FUNCTION_BLOCK "KebaHT4"	// FB 80
TITLE = Maintenance Control HT4
//
//COPYRIGHT:    (C) 1999 BY  BUEHLER AG
//                           CH-9240 UZWIL  SWITZERLAND
//
//PRODUCT:      
//
//TITLE:        MAINTENANCE MOTOR CONTROL "HT4"
//
//              LOKALE MOTOREN STEUERUNG "HT4"
//
//---------------------------------------------------------------------------
//
//IDENT:        AUTHOR:             DEPT:                         DATE:
//
//FB80.1A       S. Kalberer         CT3                           14.04.1999
//              Generated by S5/S7 Converter
//              Adjusted from S5 FB180.2C and DB180.2A
//              Outputs > 511 will set the Peripherial Output (PA) directly
//---------------------------------------------------------------------------
//
//PURPOSE:      - DATA TRANSFER BETWEEN HT4 AND PLC, VIA DB80
//
//                REMARK: ALL PASSWORD PROTECTED FUNCTIONS ARE MARKED WITH *
//
//RESTRICTIONS: - S7
//
//                !!! IMPORTANT !!!
//              - FB80 MUST BE CALLED AFTER FC9 IN OB1, TO PROCESS THE
//                OUTPUTS PROPELRY!!!
//
//              - FOLLOWING DB's MUST BE AVAILABLE:
//                . DB80 = Instance DB - COMMUNICATION BUFFER HT4 - PLC 
//                . DB81 = REFERENCE TABLE MOTORS (M)
//                . DB82 = REFERENCE TABLE VARIOUS ELEMENTS (V, FC, etc.)
//
//                . A DIGITAL OUTPUT FROM 128.0 TO 255.7 WILL BE PROCESSED
//                  INDIRECT VIA THE DB DEFINED IN DB80, DW63. THE RELEVANT
//                  DB AND DW IN THIS DB MUST BE AVAILABLE.
//                  (DW-No.IN DB = OUTPUT-BYTE-No.)
//
//              - IF THE NUMBER OF DW/OBJECT IS CHANGED, THE PARAMETERS (!@) 
//                HAVE TO BE CHANGED ACCORDINGLY !
//
//---------------------------------------------------------------------------
//$EJECT
//STRUCTURE:
//==========
//OB1:
//   | --> FC9: Call Groups
//   |
//   | --> FC80: Call Groups
//   |          |
//              |
//              | --> FB80: (REMOTE CONTROL), DB80: (COMM-BUFFER HT4 - PLC)
//                         |
//                         | --> e.g. DB81: (REF-TABLE MOTORS)
//                         |     (see Par_Motor_DBNo)
//                         | --> e.g. DB82: (REF-TABLE VARIOUS ELEMENTS)
//                         |     (see Par_Variousr_DBNo)
//       
//
//PARAMETERS and VARIABLES:
//=========================
//
//DBW 104 VAR.Errror
//  +0.0 = Error.
//  +1.0 = Error.
//  +1.1 = Error.Cfg_Fault    
//  +1.2 = Error.Obj_NoNull  
//  +1.3 = Error.Obj_Not_Found  
//  +1.4 = Error.Invalid_Password        
//  +1.5 = Error.Machine_Stop            
//  +1.6 = Error.Comm_Timeout   
//  +1.7 = Error.Summary                 
//
//DBW 106 VAR.Info
//  +0.0 = Info.Obj_Ready
//  +0.1 = Info.
//  +0.2 = Info.
//  +0.3 = Info.Obj_DO1_Set
//  +0.4 = Info.Obj_DO2_Set
//  +0.5 = Info.Obj_DO3_Set
//  +0.6 = Info.Obj_DO4_Set
//  +0.7 = Info.Obj_AO1_Set
//
//  +1.0 = Info.HT4_Enabled 
//  +1.1 = Info.HT4_Service_Mode
//  +1.2 = Info.HT4_password_ok 
//  +1.3 = Info.                
//  +1.4 = Info.                
//  +1.5 = Info.                
//  +1.6 = Info.HT4_KeyPressedFlag
//  +1.7 = Info.HT4_KeyPressedEdge
//
//DBW 108 Err_Invalid_ObjNo
//
//DBW 110 VAR_Actual_OjbNo                \
//DBW 112 VAR_DO1_ByteAddr                 | 
//DBW 114 VAR_DO1_BitAddr                  | copy from reference DB
//DBW 116 VAR_DO2_ByteAddr                 |
//DBW 118 VAR_DO2_BitAddr                  | 
//DBW 120 VAR_DO3_ByteAddr                 |
//DBW 122 VAR_DO3_BitAddr                  | 
//DBW 124 VAR_DO4_ByteAddr                 |
//DBW 126 VAR_DO4_BitAddr                  | 
//DBW 128 VAR_AO1_ByteAddr                 | 
//DBW 130 VAR_ObjState                     | 
//  +0.0 = spare                           /
//  +1.0 = ManMode
//  +1.1 = DO1_Set
//  +1.2 = DO2_Set
//  +1.3 = DO3_Set
//  +1.4 = DO4_Set
//  +1.5 = AO1_Set
//  +1.6 = 
//  +1.7 = 
//
//DBW 132 = 0    Par_AO1 Man Mode Value
//
//DBW 134 = 81  Par_Motor DB Number
//
//DBW 136 = 82  Par_Various DB Number
//
//(!@)
//DBW 138 = 0    Par_ObjDB_1stBlockOff: Byte Offset (Start oft first block)
//
//(!@)
//DBW 140 = 22   Par_ObjDB_BlockLength: Block length (Byte)
//
AUTHOR : SK
FAMILY : KebaHT4
NAME : HT4
VERSION : 1.0
VAR
  KeyStatus : STRUCT 	//Key Status
   InternalCode : BYTE ;
   UserCode : BYTE ;
   Char_8 : BOOL ;
   Char_9 : BOOL ;
   Char_A : BOOL ;
   Char_Esc : BOOL ;	//'B: esc'
   Char_C : BOOL ;
   Char_D : BOOL ;
   Char_E : BOOL ;
   Char_F : BOOL ;
   Char_F1 : BOOL ;	//'0: F1'
   Char_F2 : BOOL ;	//'1: F2'
   Char_F3 : BOOL ;	//'2: F3'
   Char_F4 : BOOL ;	//'3: F4'
   Char_F5 : BOOL ;	//'4: F5'
   Char_F6 : BOOL ;	//'5: F6'
   Char_F7 : BOOL ;	//'6: F7'
   Char_F8 : BOOL ;	//'7: F8'
   Char_O : BOOL ;
   Char_P : BOOL ;
   Char_Q : BOOL ;
   Char_R : BOOL ;
   Char_Alt : BOOL ;	//'S: Alt'
   Char_T : BOOL ;
   Char_U : BOOL ;
   Char_Start : BOOL ;	//'V: Start'
   Char_G : BOOL ;
   Char_H : BOOL ;
   Char_I : BOOL ;
   Char_J : BOOL ;
   Char_K : BOOL ;
   Char_L : BOOL ;
   Char_M : BOOL ;
   Char_N : BOOL ;
   EmergencyStop : BOOL ;
   EditModeActive : BOOL ;
   spare0602 : BOOL ;
   spare0603 : BOOL ;
   spare0604 : BOOL ;
   spare0605 : BOOL ;
   spare0606 : BOOL ;
   ActiveBit : BOOL ;
   Char_Ctrl : BOOL ;	//'W: Ctrl'
   Char_X : BOOL ;
   Char_Y : BOOL ;
   Char_Stop : BOOL ;	//'Z: Stop'
   Char_Shift : BOOL ;	//'[: Shift'
   Char_BackSlash : BOOL ;	//'\: '
   Char_SqBracketClos : BOOL ;	//']: '
   Char_Enter : BOOL ;	//'^: Enter'
  END_STRUCT ;
  EditLineNo : WORD ;	//EditLine No (HT4: 0..4)
  D_5 : WORD ;	// reserviert              ==>  S5
  D_6 : WORD ;	// reserviert              ==>  S5
  D_7 : WORD ;	// reserviert              ==>  S5
  D_8 : WORD ;	// reserviert              ==>  S5
  D_9 : WORD ;	// reserviert              <==  S5
  D_10 : WORD ;	// reserviert              <==  S5
  D_11 : WORD ;	// reserviert              <==  S5
  D_12 : WORD ;	// reserviert              <==  S5
  D_13 : WORD ;	// reserviert              <==  S5
  D_14 : WORD ;	// reserviert              <==  S5
  D_15 : WORD ;	//                         <==  S5
  DB_ID : ARRAY  [1 .. 8 ] OF CHAR ;
  LEDBitmap : STRUCT 	//LED Bitmap Red (only HT4)
   Char_8 : BOOL ;
   Char_9 : BOOL ;
   Char_A : BOOL ;
   Char_Esc : BOOL ;	//'B: esc'
   Char_C : BOOL ;
   Char_D : BOOL ;
   Char_E : BOOL ;
   Char_F : BOOL ;
   Char_F1 : BOOL ;	//'0: F1'
   Char_F2 : BOOL ;	//'1: F2'
   Char_F3 : BOOL ;	//'2: F3'
   Char_F4 : BOOL ;	//'3: F4'
   Char_F5 : BOOL ;	//'4: F5'
   Char_F6 : BOOL ;	//'5: F6'
   Char_F7 : BOOL ;	//'6: F7'
   Char_F8 : BOOL ;	//'7: F8'
   Char_O : BOOL ;
   Char_P : BOOL ;
   Char_Q : BOOL ;
   Char_R : BOOL ;
   Char_Alt : BOOL ;	//'S: Alt'
   Char_T : BOOL ;
   Char_U : BOOL ;
   Char_Start : BOOL ;	//'V: Start'
   Char_G : BOOL ;
   Char_H : BOOL ;
   Char_I : BOOL ;
   Char_J : BOOL ;
   Char_K : BOOL ;
   Char_L : BOOL ;
   Char_M : BOOL ;
   Char_N : BOOL ;
   TestOutput : BOOL ;
   SpaceLine : BOOL ;
   spare0402 : BOOL ;
   spare0403 : BOOL ;
   spare0404 : BOOL ;
   ReleaseKeyclick : BOOL ;
   DepressKeyclick : BOOL ;
   Beep : BOOL ;
   Char_Ctrl : BOOL ;	//'W: Ctrl'
   Char_X : BOOL ;
   Char_Y : BOOL ;
   Char_Stop : BOOL ;	//'Z: Stop'
   Char_Shift : BOOL ;	//'[: Shift'
   Char_BackSlash : BOOL ;	//'\: '
   Char_SqBracketClos : BOOL ;	//']: '
   Char_Enter : BOOL ;	//'^: Enter'
  END_STRUCT ;
  LEDFlashmap : STRUCT 	//LED Flashmap Red (only HT4)
   Char_8 : BOOL ;
   Char_9 : BOOL ;
   Char_A : BOOL ;
   Char_Esc : BOOL ;	//'B: esc'
   Char_C : BOOL ;
   Char_D : BOOL ;
   Char_E : BOOL ;
   Char_F : BOOL ;
   Char_F1 : BOOL ;	//'0: F1'
   Char_F2 : BOOL ;	//'1: F2'
   Char_F3 : BOOL ;	//'2: F3'
   Char_F4 : BOOL ;	//'3: F4'
   Char_F5 : BOOL ;	//'4: F5'
   Char_F6 : BOOL ;	//'5: F6'
   Char_F7 : BOOL ;	//'6: F7'
   Char_F8 : BOOL ;	//'7: F8'
   Char_O : BOOL ;
   Char_P : BOOL ;
   Char_Q : BOOL ;
   Char_R : BOOL ;
   Char_Alt : BOOL ;	//'S: Alt'
   Char_T : BOOL ;
   Char_U : BOOL ;
   Char_Start : BOOL ;	//'V: Start'
   Char_G : BOOL ;
   Char_H : BOOL ;
   Char_I : BOOL ;
   Char_J : BOOL ;
   Char_K : BOOL ;
   Char_L : BOOL ;
   Char_M : BOOL ;
   Char_N : BOOL ;
   spare0400 : BOOL ;
   spare0401 : BOOL ;
   spare0402 : BOOL ;
   spare0403 : BOOL ;
   spare0404 : BOOL ;
   spare0405 : BOOL ;
   spare0406 : BOOL ;
   spare0407 : BOOL ;
   Char_Ctrl : BOOL ;	//'W: Ctrl'
   Char_X : BOOL ;
   Char_Y : BOOL ;
   Char_Stop : BOOL ;	//'Z: Stop'
   Char_Shift : BOOL ;	//'[: Shift'
   Char_BackSlash : BOOL ;	//'\: '
   Char_SqBracketClos : BOOL ;	//']: '
   Char_Enter : BOOL ;	//'^: Enter'
  END_STRUCT ;
  TextNo_Line0 : INT ;	// Textnummer Zeile 0      <==  S5
  TextNo_Line1 : INT ;	// Textnummer Zeile 1      <==  S5
  TextNo_Line2 : INT ;	// Textnummer Zeile 2      <==  S5
  TextNo_Line3 : INT ;	// Textnummer Zeile 3      <==  S5
  D_30 : WORD ;	// reserviert              <==  S5
  D_31 : WORD ;	// reserviert              <==  S5
  D_32 : WORD ;	// reserviert              <==  S5
  D_33 : WORD ;	// reserviert              <==  S5
  D_34 : WORD ;	// Variable                <==  S5
  D_35 : WORD ;	// Variable                <==  S5
  D_36 : WORD ;	// Variable                <==  S5
  D_37 : WORD ;	// Variable                <==  S5
  D_38 : WORD ;	// Variable                <==  S5
  HT4_Inp_Password : WORD ;	// HT4.var_inp_password    <==  S5
  HT4_Target_ObjNo : WORD ;	// HT4.var_target_object_no<==> S5
  HT4_Actual_ObjNo : WORD ;	// HT4.var_actual_object_no<==> S5
  D_42 : WORD ;	// Variable                <==> S5
  D_43 : WORD ;	// Variable                <==> S5
  D_44 : WORD ;	// Variable                <==> S5
  D_45 : WORD ;	// Variable                <==> S5
  D_46 : WORD ;	// Variable                <==> S5
  D_47 : WORD ;	// Variable                <==> S5
  D_48 : WORD ;	// Variable                <==> S5
  D_49 : WORD ;	// Variable                <==> S5
  D_50 : WORD ;	// ________________________________
  D_51 : WORD ;	// ==<INTERNAL USED VARIABLES>=====
  Error : STRUCT 	// VAR.error_word
   spare0000 : BYTE ;
   spare0100 : BOOL ;
   Cfg_Fault : BOOL ;
   Obj_NoNull : BOOL ;
   Obj_NotFound : BOOL ;
   Invalid_Password : BOOL ;
   Machine_Stop : BOOL ;
   Comm_Timeout : BOOL ;
   Summary : BOOL ;
  END_STRUCT ;
  Info : STRUCT 	// VAR.info_word
   Obj_Ready : BOOL ;
   spare0001 : BOOL ;
   spare0002 : BOOL ;
   Obj_DO1_Set : BOOL ;
   Obj_DO2_Set : BOOL ;
   Obj_DO3_Set : BOOL ;
   Obj_DO4_Set : BOOL ;
   Obj_AO1_Set : BOOL ;
   HT4_Enabled : BOOL ;
   HT4_ServiceMode : BOOL ;
   HT4_PasswordOk : BOOL ;
   spare0103 : BOOL ;
   spare0104 : BOOL ;
   spare0105 : BOOL ;
   HT4_KeyPressedFlag : BOOL ;
   HT4_KeyPressedEdge : BOOL ;
  END_STRUCT ;
  Err_Invalid_ObjNo : WORD ;	// ERR.invalid_object_no
  Var_Actual_ObjNo : WORD ;	// VAR.act_object_no
  Var_DO1_ByteAddr : INT ;	// VAR.DO_1 (ByteAddress)
  Var_DO1_BitAddr : INT ;	// VAR.DO_1 (BitAddress)
  Var_DO2_ByteAddr : INT ;	// VAR.DO_2 (ByteAddress)
  Var_DO2_BitAddr : INT ;	// VAR.DO_2 (BitAddress)
  Var_DO3_ByteAddr : INT ;	// VAR.DO_3 (ByteAddress)
  Var_DO3_BitAddr : INT ;	// VAR.DO_3 (BItAddress)
  Var_DO4_ByteAddr : INT ;	// VAR.DO_4 (ByteAddress)
  Var_DO4_BitAddr : INT ;	// VAR.DO_4 (BitAddress)
  Var_AO1_ByteAddr : INT ;	// VAR.addr_AO_1 (ByteAddress)
  Var_ObjState : STRUCT 	// VAR.Obj_State
   spare0000 : BYTE ;
   ManMode : BOOL ;
   DO1_Set : BOOL ;
   DO2_Set : BOOL ;
   DO3_Set : BOOL ;
   DO4_Set : BOOL ;
   AO1_Set : BOOL ;
   spare0106 : BOOL ;
   spare0107 : BOOL ;
  END_STRUCT ;
  Par_AO1 : INT  := 250;	//* PAR.AO_1_man_mode_value_%%
  Par_Motor_DBNo : INT  := 81;	//PAR.Motor DB Number (e.g. 81)
  Par_Various_DBNo : INT  := 82;	//* PAR.Various DB Number (e.g. 82)
  Par_ObjDB_1stBlockOff : INT ;	//Object DBs: Byte Offset (Start of first block)
  Par_ObjDB_BlockLength : INT  := 22;	//Object DBs: Block length [Byte]
  spare142 : INT ;
  Var_ObjDBNo : INT ;	//Variable Actual Object DB No
  Var_ObjAR1 : DWORD ;	//Variable Actual Object Pointer
  Var_CycleTimeExt : INT ;	//TEMP.REG. CYCLE TIME EXTENSION
  spare152 : WORD  := W#16#FFFF;	//END OF FB-DATA
END_VAR
VAR_TEMP
  tmpWDBNo : WORD ;	//VAR.DB Number
  tmpDWDBPointer : DWORD ;	//VAR.Reference DB Pointer (of reference DB)
  tmpIMaxObj : INT ;	//VAR.Maximum Object of Reference DB
  tmpDWObjPointer : DWORD ;	//VAR.Object Pointer (of reference DB)
  tmpDWOutpPointer : DWORD ;	//VAR.Output Pointer
  tmpWOutpValue : WORD ;	//VAR.Output Value
  tmpILoopCnt : INT ;	//VAR.Loop Counter
  tmpIRetVal : INT ;	//VAR.Return Value
  tmpWDBLength : WORD ;	//VAR.DBLength
  tmpBWriteProt : BOOL ;	//VAR.Write Protected
END_VAR
BEGIN
NETWORK
TITLE =  INITIALIZING
      L     #KeyStatus.InternalCode;	//    int.ASCII-Code / USER-Code
      L     #KeyStatus.UserCode;	//    USER-Code
      +I;
      L     0;
      >I;
      AN    #Info.HT4_KeyPressedFlag;	//    INF.HT4_key_pressed (flag)
      =     #Info.HT4_KeyPressedEdge;	// -> INF.HT4_key_pressed (edge)
      L     #KeyStatus.InternalCode;	//    int.ASCII-Code
      L     #KeyStatus.UserCode;	//    USER-Code
      +I;
      L     0;
      >I;
      =     #Info.HT4_KeyPressedFlag;	// -> INF.HT4_key_pressed (flag)
      AN    #Info.HT4_KeyPressedEdge;	//    INF.HT4_key_pressed (edge)
      O     #Info.HT4_Enabled;	//    INF.HT4_enabled
      JC    TXT;	// ===> INITIALIZING TEXT
      S     #Info.HT4_Enabled;	// -> INF.HT4_enabled
      L     0;
      T     DIW 104;	//    VAR.error_word
TXT:  A     #Info.HT4_Enabled;	//    INF.HT4_enabled
      JC    ENAB;
      L     10;	//    WELCOME TO
      T     #TextNo_Line0;	// -> Text-No. line 0
      L     11;	//    BUHLER MOTOR
      T     #TextNo_Line1;	// -> Text-No. line 1
      L     12;	//    REMOTE CONTROL
      T     #TextNo_Line2;	// -> Text-No. line 2
      L     73;	//    Press any Key !
      T     #TextNo_Line3;	// -> Text-No. line 3
      JU    END;
// ==<HT4 ENABLED>=================
ENAB: S     #LEDBitmap.SpaceLine;	// -> Empty Line       0=<NO TEXT>
      R     #LEDBitmap.ReleaseKeyclick;	// -> Release keyklick 1=enable
      R     #LEDBitmap.DepressKeyclick;	// -> Depress keyklick 1=enable
      R     #LEDBitmap.Beep;	// -> Beep             1=on
      L     0;	// )  clear
      T     DID 40;	// )  LED Bitmap
      T     DIB 45;	// )  LED Bitmap
      T     DID 46;	// )  LED Flashmap
      T     DIB 51;	// )  LED Flashmap
      T     #TextNo_Line0;	// )  Text-No. line 0
      T     #TextNo_Line1;	// )  Text-No. line 1
      T     #TextNo_Line2;	// )  Text-No. line 2
      T     #TextNo_Line3;	// )  Text-No. line 3
END:  NOP   0;
NETWORK
TITLE =  WATCHDOG / MACHINE-STOP
      AN    #KeyStatus.ActiveBit;	//    HT4.Activ-Bit (Pass-Bit)
      L     S5T#5S;	//    monitoring time (2sec)
      SD    "SYS_T_OfflineDelay";
      A     "SYS_T_OfflineDelay";	//    HT4 - RS422-A Timeout
      =     #Error.Comm_Timeout;	// -> ERR.communication timeout
      R     #Info.HT4_Enabled;	//    INF.HT4_enabled
      A     #KeyStatus.EmergencyStop;	//    HT4.key_st.e-stop pressed
      =     #Error.Machine_Stop;	// -> ERR.machine_stop
NETWORK
TITLE =  * ENHANCED MODE
// *  --<ENABLE ENHANCED MODE>-----
      L     #KeyStatus.UserCode;	// *  USER-Code
      L     W#16#41;	// *  Taste <F1>
      ==I;	// *  IF USER-Code = 0041hex
      A     #KeyStatus.Char_Shift;	// *  HT4.key_st.shift
      S     #Info.HT4_ServiceMode;	// *->INF.HT4_enhanced_mode
      AN    #Info.HT4_ServiceMode;	// *  INF.HT4_enhanced_mode
      JC    RES;	// *
      A(;	// *  --<DISABLE ENHANCED MODE>----
      L     #KeyStatus.UserCode;	// *  USER-Code
      L     W#16#1B;	// *  Taste <ESC>
      ==I;	// *  IF USER-Code = 001Bhex
      O     #KeyStatus.Char_Esc;	// *  HT4.key_st.esc
      );	// *
      A     #KeyStatus.Char_Shift;	// *  HT4.key_st.shift
      O     #KeyStatus.EmergencyStop;	// *  HT4.key_st.e-stop pressed
      O     #Error.Comm_Timeout;	// *  ERR.communication timeout
      R     #Info.HT4_ServiceMode;	// *  INF.HT4_enhanced_mode
      JC    RES;	// *
// *  --<VERIFY PASSWORD>----------
      L     #KeyStatus.UserCode;	// *  USER-Code
      L     W#16#D;	// *  Taste <ENTER>
      ==I;	// *  IF USER-Code = 000Dhex
      A     #KeyStatus.Char_Enter;	// *  HT4.key_st.enter
      JC    PW;	// *
      JU    END3;	//END;        // *
PW:   A     #Info.HT4_PasswordOk;	// *  INF.HT4_password_ok
      JC    CLR;	// *
      L     #HT4_Inp_Password;	// *  HT4.var_inp_password
      L     W#16#1357;	// *  required password         $
      ==I;	// *
      S     #Info.HT4_PasswordOk;	// *->INF.HT4_password_ok
      R     #Info.HT4_KeyPressedEdge;	// *  INF.HT4_key_pressed (edge)
      JC    CLR;	// *
      S     #Error.Invalid_Password;	// *->ERR.invalid_password
RES:  R     #Info.HT4_PasswordOk;	// *  INF.HT4_password_ok
CLR:  L     W#16#0;	// *  clear                     $
      T     #HT4_Inp_Password;	// *  VAR.inp_password
END3: NOP   0;
NETWORK
TITLE =  DISPLAY TEXTS
      A     #Error.Summary;	//    ERR.summary
      JC    ERR1;
      AN    #Info.HT4_Enabled;	//    INF.HT4_enabled
      JC    END4;
      A     #Info.HT4_ServiceMode;	// *  INF.HT4_enhanced_mode
      JC    SERV;
// ==<NORMAL MODE>=================
//    --<SELECTION-REQUEST>--------
      A     #Info.Obj_Ready;	//    INF.obj_ready
      JC    STRT;
      L     51;	//    Please select
      T     #TextNo_Line0;	// -> Text-No. line 0
      L     64;	//    Motor No. M#####
      T     #TextNo_Line1;	// -> Text-No. line 1
      L     74;	//    Press <ENTER>
      T     #TextNo_Line2;	// -> Text-No. line 2
      JU    END4;
//    --<START-REQUEST>------------
STRT: O     #Info.Obj_DO1_Set;	//    INF.obj_DO_1_set
      O     #Info.Obj_DO2_Set;	//    INF.obj_DO_2_set
      O     #Info.Obj_DO3_Set;	//    INF.obj_DO_3_set
      O     #Info.Obj_DO4_Set;	//    INF.obj_DO_4_set
      ON    #Info.Obj_Ready;	//    INF.obj_ready
      JC    STOP;
      L     66;	//    Motor M#####
      T     #TextNo_Line0;	// -> Text-No. line 0
      L     56;	//    ready to start.
      T     #TextNo_Line1;	// -> Text-No. line 1
      L     76;	//    Press <START>
      T     #TextNo_Line2;	// -> Text-No. line 2
      JU    END4;	//END;
//    --<STOP-REQUEST>-------------
STOP: AN    #Info.Obj_DO1_Set;	//    INF.obj_DO_1_set
      AN    #Info.Obj_DO2_Set;	//    INF.obj_DO_2_set
      AN    #Info.Obj_DO3_Set;	//    INF.obj_DO_3_set
      AN    #Info.Obj_DO4_Set;	//    INF.obj_DO_4_set
      ON    #Info.Obj_Ready;	//    INF.obj_ready
      JC    END4;	//END;
      L     66;	//    Motor M#####
      T     #TextNo_Line0;	// -> Text-No. line 0
      L     57;	//    started. To stop
      T     #TextNo_Line1;	// -> Text-No. line 1
      L     77;	//    Press <STOP>
      T     #TextNo_Line2;	// -> Text-No. line 2
      JU    END4;	//END;
// ==<ENHANCED MODE>==============
// *  --<ENTER PASSWORD>-----------
SERV: A     #Info.HT4_PasswordOk;	// *  INF.HT4_password_ok
      JC    SEL;	// *
      L     13;	// *  BUHLER AG
      T     #TextNo_Line0;	// *->Text-No. line 0
      L     14;	// *  ENHANCED MODE
      T     #TextNo_Line1;	// *->Text-No. line 1
      L     61;	// *  Password ? #####
      T     #TextNo_Line2;	// *->Text-No. line 2
      L     74;	// *  Press <ENTER>
      T     #TextNo_Line3;	// *->Text-No. line 3
      JU    END4;	//END;          // *
SEL:  NOP   0;	// *  --<SELECTION-REQUEST>--------
      A     #Info.Obj_Ready;	// *  INF.obj_ready
      JC    ON;	// *
      L     51;	// *  Please select
      T     #TextNo_Line0;	// *->Text-No. line 0
      L     69;	// *  Object No.#####
      T     #TextNo_Line1;	// *->Text-No. line 1
      L     74;	// *  Press <ENTER>
      T     #TextNo_Line2;	// *->Text-No. line 2
      JU    END4;	//END;        // *
ON:   NOP   0;	// *  --<ON/OFF-REQUEST>-----------
      AN    #Info.Obj_Ready;	// *  INF.obj_ready
      JC    END4;	//END;        // *
      L     71;	// *  Object #####
      T     #TextNo_Line0;	// *->Text-No. line 0
      L     55;	// *  ready.
      T     #TextNo_Line1;	// *->Text-No. line 1
      L     82;	// *  <F7>= OFF / LN
      T     #TextNo_Line2;	// *->Text-No. line 2
      L     83;	// *  <F8>= ON  / HN
      T     #TextNo_Line3;	// *->Text-No. line 3
      JU    END4;	//END;
// ==<ERROR-TEXTS>=================
ERR1: AN    #Error.Cfg_Fault;	//    ERR.cfg_fault
      JC    ERR2;
      L     21;	//    **** ERROR *****
      T     #TextNo_Line0;	// -> Text-No. line 0
      L     22;	//    CONFIG. FAULT
      T     #TextNo_Line1;	// -> Text-No. line 1
      JU    ESC;
ERR2: AN    #Error.Obj_NoNull;	//    ERR.object_no_<=null
      JC    ERR3;
      L     21;	//    **** ERROR *****
      T     #TextNo_Line0;	// -> Text-No. line 0
      L     23;	//    INVALID No.00000
      T     #TextNo_Line1;	// -> Text-No. line 1
      JU    ESC;
ERR3: AN    #Error.Obj_NotFound;	//    ERR.object_not_found
      JC    ERR4;
      A     #Info.HT4_ServiceMode;	// *  INF.HT4_enhanced_mode
      L     70;	//    Object No. #####
      JC    TXL0;
      L     65;	//    Motor No. M#####
TXL0: T     #TextNo_Line0;	// -> Text-No. line 0
      L     53;	//    not found in PLC
      T     #TextNo_Line1;	// -> Text-No. line 1
      L     54;	//    Try again
      T     #TextNo_Line2;	// -> Text-No. line 2
      JU    ESC;
ERR4: AN    #Error.Invalid_Password;	// *  ERR.invalid_password
      JC    ERR5;	// *
      L     21;	// *  **** ERROR *****
      T     #TextNo_Line0;	// *->Text-No. line 0
      L     28;	// *  INVALID PASSWORD
      T     #TextNo_Line1;	// *->Text-No. line 1
      JU    ESC;
ERR5: AN    #Error.Machine_Stop;	//    ERR.machine_stop
      ON    #Info.HT4_Enabled;	//    INF.HT4_enabled
      JC    END4;	//END;
      L     21;	//    **** ERROR *****
      T     #TextNo_Line0;	// -> Text-No. line 0
      L     26;	//    MACHINE-STOP
      T     #TextNo_Line1;	// -> Text-No. line 1
      L     27;	//    PRESSED
      T     #TextNo_Line2;	// -> Text-No. line 2
      A     #KeyStatus.EmergencyStop;	//    HT4.key_st.e-stop pressed
      JC    END4;	//END;
ESC:  L     75;	//    Press <ESC>
      T     #TextNo_Line3;	// -> Text-No. line 3
END4: NOP   0;
NETWORK
TITLE =  KEYBOARD LED's
      A     #KeyStatus.EmergencyStop;	//    HT4.key_st.e-stop pressed
      ON    #Info.HT4_Enabled;	//    INF.HT4_enabled
      JC    END5;	//END;
      A     #Error.Summary;	//    ERR.summary
      S     #LEDFlashmap.Char_Esc;	// -> LED Flashmap (ESC)
      JC    END5;	//END;
      A     #Info.Obj_Ready;	//    INF.obj_ready
      AN    #Info.Obj_DO1_Set;	//    INF.obj_DO_1_set
      AN    #Info.Obj_DO2_Set;	//    INF.obj_DO_2_set
      AN    #Info.Obj_DO3_Set;	//    INF.obj_DO_3_set
      AN    #Info.Obj_DO4_Set;	//    INF.obj_DO_4_set
      S     #LEDBitmap.Char_Stop;	// -> LED Bitmap (STOP)
      A     #Info.Obj_Ready;	//    INF.object_ready
      AN    #Info.HT4_ServiceMode;	// *  INF.HT4_enhanced_mode
      A(;
      O     #Info.Obj_DO1_Set;	//    INF.obj_DO_1_set
      O     #Info.Obj_DO2_Set;	//    INF.obj_DO_2_set
      O     #Info.Obj_DO3_Set;	//    INF.obj_DO_3_set
      O     #Info.Obj_DO4_Set;	//    INF.obj_DO_4_set
      );
      S     #LEDBitmap.Char_Start;	// -> LED Bitmap (START)
//xx add Obj_DO3/4
      A     #Info.HT4_ServiceMode;	// *  INF.HT4_enhanced_mode
      A     #Info.Obj_DO1_Set;	//    INF.obj_DO_1_set
      S     #LEDBitmap.Char_F7;	// -> LED Bitmap (F7)
      A     #Info.HT4_ServiceMode;	// *  INF.HT4_enhanced_mode
      A     #Info.Obj_DO2_Set;	//    INF.obj_DO_2_set
      S     #LEDBitmap.Char_F8;	// -> LED Bitmap (F8)
END5: NOP   0;
NETWORK
TITLE =  SEARCH OBJECT
      A     #Error.Summary;	//    ERR.summary 
      ON    #Info.HT4_Enabled;	//    INF.HT4_enabled
      ON    #Info.HT4_KeyPressedEdge;	//    INF.HT4_key_pressed (edge)
      JC    END6;	//END;
// --<ENTER>-----------------------
      L     #KeyStatus.UserCode;	//    USER-Code
      L     W#16#D;	//    Taste <ENTER>
      <>I;	//    IF USER-Code = 000Dhex
      ON    #KeyStatus.Char_Enter;	//    HT4.key_st.enter
      JC    END6;	//END;
      AN    #Info.HT4_ServiceMode;	// *  INF.HT4_enhanced_mode
      L     #Par_Motor_DBNo;	// Standard: Motor-DB
      JC    DB;
      AN    #Info.HT4_PasswordOk;	// *  INF.HT4_password_ok
      L     #Par_Various_DBNo;	// Standard: Various-DB
      JC    END6;	//END;
DB:   T     #tmpWDBNo;	//Save DB-Number 
      CALL  "SIEMENS_TEST_DB" (
           DB_NUMBER                := #tmpWDBNo,
           RET_VAL                  := #tmpIRetVal,
           DB_LENGTH                := #tmpWDBLength,
           WRITE_PROT               := #tmpBWriteProt);	//Check DB
      L     W#16#0;	// RET_VAL <>0: Cfg-Error_1
      L     #tmpIRetVal;
      <>I;
      JC    ER61;	// ==> ERROR_1
      OPN   DB [#tmpWDBNo];	// -> Open Reference DB
// ________________________________
      L     0;	// ** clear **
      T     #Var_Actual_ObjNo;	// -> VAR.act_object_no
// --------------------------------
      L     W#16#0;	// $
      L     #HT4_Target_ObjNo;	//    HT4_var.target_object_no
      ==I;	// 2B: IF object_no Zero
      JC    ER62;	// ==> ERROR_2
// --<SEARCH OBJECT>---------------
      L     DBLG;	// )   lenght DB
      L     #Par_ObjDB_1stBlockOff;	// )    - reserved bytes
      -D;
      L     #Par_ObjDB_BlockLength;	// )    Blocklength
      /D;	// )   
      T     #tmpIMaxObj;	// )-->max_Object
ZYK1: T     #tmpILoopCnt;	//Calculate AR1 address
      +     -1;
      L     #Par_ObjDB_BlockLength;	// )   Blocklength
      *D;
      L     #Par_ObjDB_1stBlockOff;	// )   - reserved bytes
      +D;
      SLD   3;	//Get pointer address
      LAR1;
      L     DBW [AR1,P#0.0];	//Save temporary low word
      L     #HT4_Target_ObjNo;	// )  HT4_var.target_object_no
      ==I;	// )  IF object_no found ?
      JC    FOUN;	// )
      L     #tmpILoopCnt;
      LOOP  ZYK1;
      JU    ER63;	// ==> ERROR_3
// --<OBJECT FOUND>----------------
FOUN: T     #HT4_Actual_ObjNo;	// )->HT4_var.actual_object_no
      T     #Var_Actual_ObjNo;	// )->VAR.act_object_no
// Save AR1 Register with Pointer to actual Object
      TAR1;
      T     #Var_ObjAR1;
      L     DBNO;
      T     #Var_ObjDBNo;
// Read DO_1 Byte/BitAddress
      L     DBW [AR1,P#2.0];	// VAR_DO_1_ByteAddr
      T     #Var_DO1_ByteAddr;
      L     DBW [AR1,P#4.0];	// VAR_DO_1_BitAddr
      T     #Var_DO1_BitAddr;
// Read DO_2 Byte/BitAddress
      L     DBW [AR1,P#6.0];	// VAR_DO_2_ByteAddr
      T     #Var_DO2_ByteAddr;
      L     DBW [AR1,P#8.0];	// VAR_DO_2_BitAddr
      T     #Var_DO2_BitAddr;
// Read DO_3 Byte/BitAddress
      L     DBW [AR1,P#10.0];	// VAR_DO_3_ByteAddr
      T     #Var_DO3_ByteAddr;
      L     DBW [AR1,P#12.0];	// VAR_DO_3_BitAddr
      T     #Var_DO3_BitAddr;
// Read DO_4 Byte/BitAddress
      L     DBW [AR1,P#14.0];	// VAR_DO_4_ByteAddr
      T     #Var_DO4_ByteAddr;
      L     DBW [AR1,P#16.0];	// VAR_DO_4_BitAddr
      T     #Var_DO4_BitAddr;
// Read AO ByteAddress
      L     DBW [AR1,P#18.0];	// VAR_AO_1_ByteAddr
      T     #Var_AO1_ByteAddr;
// Read Object State
      L     DBW [AR1,P#20.0];	// VAR_Obj_State
      T     DIW 126;	//Var_ObjState
// --<TESTS>-----------------------
      L     #Var_DO1_ByteAddr;
      L     #Var_DO1_BitAddr;
      +I;
      L     0;
      <=I;	//    IF DO_1 = 0,0
      A(;
      L     #Var_DO2_ByteAddr;
      L     #Var_DO2_BitAddr;
      +I;
      L     0;
      <=I;	//    IF DO_2 = 0,0
      );
      A(;
      L     #Var_DO3_ByteAddr;
      L     #Var_DO3_BitAddr;
      +I;
      L     0;
      <=I;	//    IF DO_3 = 0,0
      );
      A(;
      L     #Var_DO4_ByteAddr;
      L     #Var_DO4_BitAddr;
      +I;
      L     0;
      <=I;	//    IF DO_4 = 0,0
      );
      JC    ER61;	// ===> NO INPUT DEFINED
      L     #Var_DO1_BitAddr;	//    VAR.bit_addr_DO_1
      L     7;
      >I;	//    IF bit_addr > 7
      O(;
      L     #Var_DO2_BitAddr;	//    VAR.bit_addr_DO_2
      L     7;
      >I;	//    IF bit_addr > 7
      );
      O(;
      L     #Var_DO3_BitAddr;	//    VAR.bit_addr_DO_3
      L     7;
      >I;	//    IF bit_addr > 7
      );
      O(;
      L     #Var_DO4_BitAddr;	//    VAR.bit_addr_DO_4
      L     7;
      >I;	//    IF bit_addr > 7
      );
      JC    ER61;	// ===> INVALID BIT ADDRESS
      A(;
      L     #Var_DO1_ByteAddr;	//    VAR.byte_addr_DO_1
      L     511;
      >I;	//    IF byte_addr. > 511
      O(;
      L     #Var_DO2_ByteAddr;	//    VAR.byte_addr_DO_2
      L     511;
      >I;	//    IF byte_addr. > 511
      );
      O(;
      L     #Var_DO3_ByteAddr;	//    VAR.byte_addr_DO_3
      L     511;
      >I;	//    IF byte_addr. > 511
      );
      O(;
      L     #Var_DO4_ByteAddr;	//    VAR.byte_addr_DO_4
      L     511;
      >I;	//    IF byte_addr. > 511
      );
      );
      JC    ER61;	// ===> DB0 = INVALID DB
      S     #Info.Obj_Ready;	// -> INF.obj_ready
      S     #Var_ObjState.ManMode;	// -> INF.obj_man_mode
      JU    END6;	//END;
ER61: NOP   0;	// --<ERROR ROUTINE>---------------
      S     #Error.Cfg_Fault;	// -> ERR.cfg_fault
      JU    END6;	//END;
ER62: S     #Error.Obj_NoNull;	// -> ERR.object_no_<=null
      JU    END6;	//END;
ER63: S     #Error.Obj_NotFound;	// -> ERR.object_not_found
      L     #HT4_Target_ObjNo;	//    HT4_var.target_object_no
      T     #Err_Invalid_ObjNo;	// -> invalid_object_no
      JU    END6;	//END;
END6: NOP   0;
NETWORK
TITLE =  MOTOR CONTROL ON_1 / ON_2
      AN    #Info.Obj_Ready;	//    INF.obj_ready
      O     #Info.HT4_ServiceMode;	// *  INF.HT4_enhanced_mode
      JC    END7;	//END;
// --<MOTOR ON_1>-----------------
      L     #KeyStatus.UserCode;	//    USER-Code
      L     W#16#4C;	//    Taste <Start>
      ==I;	//    IF USER-Code = 004Chex
      A     #KeyStatus.Char_Start;	//    HT4.key_st.start
      AN    #KeyStatus.Char_Shift;	//    HT4.key_st.shift (reverse)
      AN    #Info.Obj_DO2_Set;	//    INF.obj_DO_2_set
      S     #Info.Obj_DO1_Set;	// -> INF.obj_DO_1_set
// --<MOTOR ON_2>-----------------
      L     #KeyStatus.InternalCode;	//    ASCII-Code
      L     W#16#56;	//    Taste <Start>
      ==I;	//    IF USER-Code = 0056hex
      A     #KeyStatus.Char_Start;	//    HT4.key_st.start
      A     #KeyStatus.Char_Shift;	//    HT4.key_st.shift (reverse)
      AN    #Info.Obj_DO1_Set;	//    INF.obj_DO_1_set
      S     #Info.Obj_DO2_Set;	// -> INF.obj_DO_2_set
END7: NOP   0;
NETWORK
TITLE =  * VARIOUS CONTROL ON_1 / ON_2
      AN    #Info.Obj_Ready;	// *  INF.obj_ready
      ON    #Info.HT4_PasswordOk;	// *  INF.HT4_password_ok
      JC    END8;	//END;        // *
// --<OBJECT ON_1>-----------------
      L     #KeyStatus.UserCode;	// *  USER-Code
      L     W#16#47;	// *  Taste <F7> (on,hn,open)
      ==I;	// *  IF USER-Code = 0047hex
      A     #KeyStatus.Char_F7;	// *  HT4.key_st.F7
      S     #Info.Obj_DO1_Set;	// *->INF.obj_DO_1_set
      R     #Info.Obj_DO2_Set;	// *  INF.obj_DO_2_set
// --<OBJECT ON_2>-----------------
      L     #KeyStatus.UserCode;	// *  USER-Code
      L     W#16#48;	// *  Taste <F8> (off, ln)
      ==I;	// *  IF USER-Code = 0048hex
      A     #KeyStatus.Char_F8;	// *  HT4.key_st.F8
      S     #Info.Obj_DO2_Set;	// *->INF.obj_DO_2_set
      R     #Info.Obj_DO1_Set;	// *  INF.obj_DO_1_set
END8: NOP   0;
NETWORK
TITLE =  ESC, MACHINE-STOP, OFF
// --<ESC OBJECT>------------------
      L     #KeyStatus.UserCode;	// *  USER-Code
      L     W#16#41;	// *  Taste <F1>
      ==I;	// *  IF USER-Code = 0041hex
      A     #KeyStatus.Char_Shift;	// *  HT4.key_st.shift
      O(;
      L     #KeyStatus.UserCode;	//    USER-Code
      L     W#16#1B;	//    Taste <ESC>
      ==I;	//    IF USER-Code = 001Bhex
      );
      O     #KeyStatus.Char_Esc;	//    HT4.key_st.esc
      JC    ESC9;	//ESC;
// --<MACHINE-STOP>----------------
      A     #KeyStatus.EmergencyStop;	//    HT4.key_st.e-stop pressed
      O     "SYS_T_OfflineDelay";	//    HT4 - RS422-A Timeout
      ON    #Info.HT4_Enabled;	//    INF.HT4_enabled 
      JC    ESC9;	//ESC;
// --<OBJECT OFF>------------------
      L     #KeyStatus.UserCode;	//    USER-Code
      L     W#16#4F;	//    Taste <Stop>
      ==I;	//    IF USER-Code = 004Fhex
      O     #KeyStatus.Char_Stop;	//    HT4.key_st.stop
      JC    OFF;
      JU    END9;	//END;
// --<RESET FUNCTIONS>-------------
ESC9: L     W#16#0;	// $
      T     #HT4_Actual_ObjNo;	// -> reset HT4_var.act_obj_no
      T     #Err_Invalid_ObjNo;	// -> reset ERR.invalid_object_no
      T     #Var_Actual_ObjNo;	// -> reset VAR.act_obj_no
      L     DIW 104;	//    VAR.error_word
      L     2#1100000;	//    0 = reset
      AW;
      T     DIW 104;	// -> reset VAR.error_word
      SET;
      R     #Info.Obj_Ready;	// -> reset INF.obj_ready
      R     #Info.Obj_DO1_Set;	// -> reset INF.obj_DO_1_set
      R     #Info.Obj_DO2_Set;	// -> reset INF.obj_DO_2_set
      R     #Info.Obj_DO3_Set;	// -> reset INF.obj_DO_3_set
      R     #Info.Obj_DO4_Set;	// -> reset INF.obj_DO_4_set
      R     #Info.Obj_AO1_Set;	// -> reset INF.obj_AO_1_set
// --<OUTPUTS OFF >----------------
OFF:  SET;
      R     #Info.Obj_DO1_Set;	// -> reset INF.obj_DO_1_set
      R     #Info.Obj_DO2_Set;	// -> reset INF.obj_DO_2_set
      R     #Info.Obj_DO3_Set;	// -> reset INF.obj_DO_3_set
      R     #Info.Obj_DO4_Set;	// -> reset INF.obj_DO_4_set
END9: NOP   0;
NETWORK
TITLE =  CONTROL DIGITAL OUTPUT 1
      A     #Error.Cfg_Fault;	//    ERR.cfg_fault
      JC    ED10;	//END;
      L     #Var_DO1_ByteAddr;	//    VAR.Byteaddr_DO_1
      L     #Var_DO1_BitAddr;	//    VAR.Bitaddr_DO_1
      +I;
      L     0;
      <=I;	//    IF DO_1 = 0,0
      R     #Info.Obj_DO1_Set;	//    INF.obj_DO_1_set
      JC    ED10;	//END;
      L     #Var_DO1_ByteAddr;	//    VAR.byte_addr_DO_1
      L     511;
      >I;	//    IF byte_addr. > 511
      JC    PA10;	//DB;
// --<DO_1 <= 511.7>-------------
      A     #Info.Obj_DO1_Set;	//    INF.obj_DO_1_set
      L     #Var_DO1_ByteAddr;	//    VAR.Byteaddr_DO_1
      SLW   3;
      L     #Var_DO1_BitAddr;	//    VAR.Bitaddr_DO_1
      SLW   5;
      SRW   5;
      OW;
      T     #tmpDWOutpPointer;
      =     Q [#tmpDWOutpPointer];	// -> DO_1 ON    [ <= DO 511.7]
      JU    ED10;	//END;
// --<DO_1 > 511.7>--------------
PA10: L     #Var_DO1_ByteAddr;	//    VAR.Byteaddr_DO_1
      SLW   3;
      T     #tmpDWOutpPointer;
      L     DBB [#tmpDWOutpPointer];	// -> act. DB_DO.DBB (DO 7....0)
      T     #tmpWOutpValue;
      A     #Info.Obj_DO1_Set;	// )   INF.DO_1_set
      JCN   ED10;
      L     #Var_DO1_BitAddr;	// ) Set bit
      L     1;
      SLW;
      L     #tmpWOutpValue;
      OW;
      T     PQB [#tmpDWOutpPointer];	// -> act. DB_DO.DBB (DO 7....0)
ED10: NOP   0;
NETWORK
TITLE =  CONTROL DIGITAL OUTPUT 2
      A     #Error.Cfg_Fault;	//    ERR.cfg_fault
      JC    ED11;	//END;
      L     #Var_DO2_ByteAddr;	//    VAR.Byteaddr_DO_2
      L     #Var_DO2_BitAddr;	//    VAR.Bitaddr_DO_2
      +I;
      L     0;
      <=I;	//    IF DO_1 = 0,0
      R     #Info.Obj_DO2_Set;	//    INF.obj_DO_2_set
      JC    ED11;	//END;
      L     #Var_DO2_ByteAddr;	//    VAR.byte_addr_DO_2
      L     511;
      >I;	//    IF byte_addr. > 511
      JC    PA11;	//DB;
// --<DO_1 <= 511.7>-------------
      A     #Info.Obj_DO2_Set;	//    INF.obj_DO_2_set
      L     #Var_DO2_ByteAddr;	//    VAR.Byteaddr_DO_2
      SLW   3;
      L     #Var_DO2_BitAddr;	//    VAR.Bitaddr_DO_2
      SLW   5;
      SRW   5;
      OW;
      T     #tmpDWOutpPointer;
      =     Q [#tmpDWOutpPointer];	// -> DO_2_ON    [ <= DO 511.7]
      JU    ED11;	//END;
// --<DO_2 > 511.7>--------------
PA11: L     #Var_DO2_ByteAddr;	//    VAR.Byteaddr_DO_2
      SLW   3;
      T     #tmpDWOutpPointer;
      L     DBB [#tmpDWOutpPointer];	// -> act. DB_DO.DBB (DO 7....0)
      T     #tmpWOutpValue;
      A     #Info.Obj_DO2_Set;	// )   INF.DO_2_set
      JCN   ED11;
      L     #Var_DO2_BitAddr;	// ) Set bit
      L     1;
      SLW;
      L     #tmpWOutpValue;
      OW;
      T     PQB [#tmpDWOutpPointer];	// -> act. DB_DO.DBB (DO 7....0)
ED11: NOP   0;
NETWORK
TITLE =  CONTROL ANALOG OUTPUT 1
      A     #Error.Cfg_Fault;	//    ERR.cfg_fault
      JC    ED12;	//END;
      L     #Var_AO1_ByteAddr;	//    VAR.addr_AO_1
      L     0;
      <=I;	//    IF DO_1 = 0,0
      ON    #Var_ObjState.ManMode;	//    INF.obj_man_mode
      R     #Info.Obj_AO1_Set;	//    INF.obj_AO_1_set
      JC    ED12;	//END;
// Calculate Output address offset
      A     #Info.Obj_Ready;	// )  INF.obj_ready
      =     #Info.Obj_AO1_Set;	// )->INF.obj_AO_1_set
      JC    VALU;
      L     0;	//  )
      JU    RE12;	//  )===> clear AO
VALU: L     #Par_AO1;	// )  PAR.AO_1_man_mode_value_%%
RE12: T     #tmpWOutpValue;	// -> AO_1
      L     511;
      L     #Var_AO1_ByteAddr;	//    VAR.Byteaddr_AO_1
      <=I;	//    IF byte_addr. > 511
      SLW   3;	//Get Bit-Address
      T     #tmpDWOutpPointer;
      JC    PA12;	//DB;
// --<AO_1 <= 511>-------------
      L     #tmpWOutpValue;
      T     QW [#tmpDWOutpPointer];	// -> AO_1    [ <= AO 511]
      JU    ED12;	//END;
// --<AO_1 > 511>--------------
PA12: L     #tmpWOutpValue;
      T     PQW [#tmpDWOutpPointer];	// -> act. DB_DO.DBB (AO >511)
ED12: NOP   0;
NETWORK
TITLE =  ERROR SUMMARY
      L     DIW 104;	//    VAR.error_word
      L     2#1111111;
      AW;
      L     0;
      >I;
      =     #Error.Summary;	// -> ERR.summary
      R     #Info.Obj_Ready;	// -> reset INF.obj_ready
NETWORK
TITLE =  INITIALIZING
      A     #Error.Cfg_Fault;	// )  ERR.cfgFault
      ON    #Var_ObjState.ManMode;	// )  INF.obj_man_mode
      JC    RE14;	//RES;        // )
      AN    #Info.Obj_Ready;	// )  INF.obj_ready
      R     #Var_ObjState.ManMode;	// )->reset INF.obj_man_mode
      A     #Info.Obj_DO1_Set;	// )  INF.obj_DO_1_set
      =     #Var_ObjState.DO1_Set;	// )->
      A     #Info.Obj_DO2_Set;	// )  INF.obj_DO_2_set
      =     #Var_ObjState.DO2_Set;	// )->
      A     #Info.Obj_DO3_Set;	// )  INF.obj_DO_3_set
      =     #Var_ObjState.DO3_Set;	// )->
      A     #Info.Obj_DO4_Set;	// )  INF.obj_DO_4_set
      =     #Var_ObjState.DO4_Set;	// )->
      A     #Info.Obj_AO1_Set;	// )  INF.obj_AO_1_set
      =     #Var_ObjState.AO1_Set;	// )->
      L     #Var_ObjDBNo;
      T     #tmpWDBNo;
      OPN   DB [#tmpWDBNo];
      L     #Var_ObjAR1;	// )  Abs.Address of act. Object
      LAR1;
      L     DIW 126;	// )  obj_status
      T     DBW [AR1,P#20.0];	// )-> Object_State
RE14: A     #Info.Obj_Ready;	//    INF.obj_ready
      JC    ED14;	//END;
      L     0;	// )
      T     DIB 106;	// )-> reset VAR.info_byte
      T     #Var_DO1_ByteAddr;
      T     #Var_DO2_ByteAddr;
      T     #Var_DO3_ByteAddr;
      T     #Var_DO4_ByteAddr;
      T     #Var_DO1_BitAddr;
      T     #Var_DO2_BitAddr;
      T     #Var_DO3_BitAddr;
      T     #Var_DO4_BitAddr;
      T     #Var_AO1_ByteAddr;
      T     DIW 126;	// -> reset Var_ObjState
ED14: SET;
      R     #KeyStatus.ActiveBit;	// -> reset HT4.Activ-Bit
NETWORK
TITLE =  CYCLE TIME EXTENSION
      A     "SYS_infLog1";
      BEC;	// !! USED IF ONLY MAINTENANCE
LOOP: L     #Var_CycleTimeExt;	//    MOTOR CONTROL SOFTWARE
      +     1;	//    INSTALLED IN PLC !!
      T     #Var_CycleTimeExt;
      L     25000;
      <I;
      JC    LOOP;
      L     0;
      T     #Var_CycleTimeExt;
END_FUNCTION_BLOCK

FUNCTION_BLOCK "GCS7_M_RGRP"	// FB 81
TITLE = Machine RGRP PRIMUS
//  
//COPYRIGHT:    (C) 2004  BUHLER AG, CH-9240 UZWIL,  SWITZERLAND
//
//PRODUCT:      GCS7
//
//TITLE:        FB 81 MACHINE-CONTROL:RGRP PRIMUS
//-------------------------------------------------------------------------
//
//IDENT:        AUTHOR:             DEPT:                       DATE:
//FB81.1.1      A.Egli              CT3                         11-Sep-2007
//              Monitoring LSSieve only if MotorSieve is started
//FB81.1.0      A.Egli              CT3                         04-Aug-2004
//              1st Release in S7
//
//-------------------------------------------------------------------------
//
//PURPOSE:      MANUAL : see [LL.RGRPxxMAN]
//
//RESTRICTIONS: S7
//
//-------------------------------------------------------------------------
//
AUTHOR : EA
FAMILY : GCS7LL
NAME : RGRP
VERSION : 1.1
VAR
  Ma : UDT 20810;
  LS1Sieve : FB 14;	//Element
  LS2Sieve : FB 14;	//Element
  FlapLower : FB 20;	//Element
  FlapUpper : FB 20;	//Element
  MotorSieve : FB 12;	//Element
  PosFlapAir : FB 20;	//Element
  MotorFlapAir : FB 12;
  PosFlapFeed : FB 20;	//Element
  MotorFlapFeed : FB 12;
  Airlock : FB 12;	//Element
  FeedRoll : FB 12;	//Element
  FlowDetector : FB 19;	//Element
  Fan1 : FB 12;	//Element
  Fan2 : FB 12;	//Element
END_VAR
VAR_TEMP
  tmpFaultSum : BOOL ;
  tmpLocal : BOOL ;
  tmpEnable : BOOL ;
  tmpStartReq : BOOL ;
  tmpLenDyn : INT ;
  tmpBit : BOOL ;
  tmpEnableVender : BOOL ;
  tmpNext : BOOL ;
  tmpStarted : BOOL ;
  tmpStopped : BOOL ;
  tmpWaySieveAdjusted : BOOL ;
  tmpFlapVendorAdjusted : BOOL ;
  tmpToHigh : BOOL ;
  tmpFactor : REAL ;
  tmpSeqStop : BOOL ;
END_VAR
BEGIN
NETWORK
TITLE =
      L     60;
      T     #tmpLenDyn;
NETWORK
TITLE = PC Control
//=== Test Object number =====================
      L     "SYS_DirectCtrlDB".PC.ObjectNo;	//PCControl.ObjectNo
      L     #Ma.Par.ParObjectNo;	//Input ObjectNo
      <>I;
      JC    aEnd;
//=== Test OType      ========================
      L     2081;	//Input object type
      L     "SYS_DirectCtrlDB".PC.ObjectType;	//PCControl.ObjectType
      <>I;
      JC    aEnd;
//=== Test Handshake =========================
      A     "SYS_DirectCtrlDB".PC.Hsk.FExamine;	// Handshake.FExamine
      JC    aExa;
      A     "SYS_DirectCtrlDB".PC.Hsk.FDefineCmd;	// Handshake.FDefineCmd
      JC    aCmd;
      A     "SYS_DirectCtrlDB".PC.Hsk.FDefinePara;	// Handshake.FDefinePara
      JC    pPar;
aIni: L     2;	// FcInit
      UC    "SYS_DirectCtrl";
      JU    aEnd;
// Write parameter 
pPar: LAR1  P#DBX 58.0;
      L     P#30.0;
      +AR1;
      L     DBW [AR1,P#4.0];
      T     #Ma.Par.ParClearingTime;
// Write new commands from PC to Interface of group 
aCmd: A     "SYS_DirectCtrlDB".PC.Cmd1[8];	//Cmd1[8]=CmdOff
      S     #Ma.CmdOff;
      R     #Ma.OutStartReqMan;
      A     "SYS_DirectCtrlDB".PC.Cmd1[9];	//Cmd1[9]=CmdOn
      S     #Ma.CmdOn;
      S     #Ma.OutStartReqMan;
      A     "SYS_DirectCtrlDB".PC.Cmd1[6];	//Cmd1[6]=CmdNewJob
      S     #Ma.CmdNewJob;
      A     "SYS_DirectCtrlDB".PC.Cmd1[10];	//Cmd1[10]=CmdNext
      S     #Ma.CmdNext;
      A     "SYS_DirectCtrlDB".PC.Cmd1[11];	//Cmd1[11]=CmdFaultReset
      S     #Ma.CmdFaultReset;
      A     "SYS_DirectCtrlDB".PC.Cmd1[13];	//Cmd1[13]=CmdManualOn
      S     #Ma.InManual;
      A     "SYS_DirectCtrlDB".PC.Cmd2[13];	//Cmd2[13]=CmdManualOff
      R     #Ma.InManual;
      R     #Ma.OutStartReqMan;
      JU    aIni;
aExa: TAR2;	// Address dynamic data
      T     "SYS_DirectCtrlDB".GC.InDynAddr;	// -->PCControl.GC.InDynAddr
      L     #tmpLenDyn;	// Length Dynamic data
      T     "SYS_DirectCtrlDB".GC.InDynLen;	// -->PCControl.GC.InDynLen
      L     0;
      T     "SYS_DirectCtrlDB".GC.InParaAddr;	// -->PCControl.GC.InParaAddr
      T     "SYS_DirectCtrlDB".GC.InParaLen;	// -->PCControl.GC.InParaLen
      L     1;	// Code FcExamine
      UC    "SYS_DirectCtrl";
      L     10;	//Revision
      T     "SYS_DirectCtrlDB".GC.Revision;
aEnd: NOP   0;
NETWORK
TITLE = Interlocking
//===Global Group Orders===
      A     "GCS7_Gr_OutManualOn";	//Gr.OutManualOn
      S     #Ma.InManual;
      A     "GCS7_Gr_OutManualOff";	//Gr.OutManualOff
      R     #Ma.InManual;
      A     #Ma.InManual;
      S     "GCS7_Gr_InManual";	//Gr.InManual
      A     #Ma.InLocal;
      AN    #Ma.InManual;
      =     #tmpLocal;
      A     #Ma.InSeqStop;
      AN    #Ma.InManual;
      =     #tmpSeqStop;
      A     #Ma.InManual;
      R     #Ma.InClearing;
//--- Fault----
      A     #LS1Sieve.StFault;
      O     #LS2Sieve.StFault;
      O     #FlapLower.StFault;
      O     #FlapUpper.StFault;
      O     #MotorSieve.StFault;
      O     #PosFlapAir.StFault;
      O     #PosFlapFeed.StFault;
      O     #Airlock.StFault;
      O     #FeedRoll.StFault;
      O     #FlowDetector.OutFaulted;
      O     #Fan1.StFault;
      O     #Fan2.StFault;
      O     #MotorFlapAir.StFault;
      O     #MotorFlapFeed.StFault;
      =     #tmpFaultSum;
//--- OutCleared----
      AN    #Ma.InClearing;
      R     #Ma.OutCleared;
//--- Temporare----
      AN    #Ma.CmdOff;
      A     #Ma.InEnable;
      A(;
      AN    #Ma.InClearing;
      ON    #Ma.OutCleared;
      );
      AN    #Ma.InManual;
      O;
      A     #Ma.InManual;
      A     #Ma.OutStartReqMan;
      =     #tmpEnable;
      AN    #Ma.InManual;
      A     #Ma.CmdNext;
      O;
      A     #Ma.InManual;
      A     #Ma.OutStartReqMan;
      =     #tmpNext;
//--- Local mode --
      A     #tmpLocal;
      =     #LS1Sieve.InLocal;
      =     #LS2Sieve.InLocal;
      =     #FlapLower.InLocal;
      =     #FlapUpper.InLocal;
      =     #MotorSieve.InLocal;
      =     #Airlock.InLocal;
      =     #FeedRoll.InLocal;
      =     #FlowDetector.InLocal;
      =     #Fan1.InLocal;
      =     #Fan2.InLocal;
//--- Fault Reset -------------
      A     #Ma.CmdFaultReset;
      S     #LS1Sieve.CmdFaultReset;
      S     #LS2Sieve.CmdFaultReset;
      S     #FlapLower.CmdFaultReset;
      S     #FlapUpper.CmdFaultReset;
      S     #MotorSieve.CmdFaultReset;
      S     #Airlock.CmdFaultReset;
      S     #FeedRoll.CmdFaultReset;
      S     #FlowDetector.CmdFaultReset;
      S     #Fan1.CmdFaultReset;
      S     #Fan2.CmdFaultReset;
      A     #Ma.InpAirMinus;
      O     #Ma.InpAirPlus;
      O     #Ma.InpFeedMinus;
      O     #Ma.InpFeedPlus;
      FP    #Ma.Par.tmpEdgeInpLocal;
      O     #Ma.CmdFaultReset;
      S     #PosFlapAir.CmdFaultReset;
      S     #MotorFlapAir.CmdFaultReset;
      S     #PosFlapFeed.CmdFaultReset;
      S     #MotorFlapFeed.CmdFaultReset;
NETWORK
TITLE = Interlocking Sieve
//--- Monitoring
      A     #MotorSieve.StStartedFwd;	//[1.1]
      =     #LS1Sieve.InMonTrue;
      =     #LS2Sieve.InMonTrue;
//--- FlapLower----
      L     #Ma.InPosFlapLower;
      L     1;
      ==I;
      =     #FlapLower.InLN;
      L     #Ma.InPosFlapLower;
      L     2;
      ==I;
      =     #FlapLower.CmdMiddle1;
      L     #Ma.InPosFlapLower;
      L     3;
      ==I;
      =     #FlapLower.CmdHN;
//--- FlapUpper----
      L     #Ma.InPosFlapUpper;
      L     1;
      ==I;
      =     #FlapUpper.InLN;
      L     #Ma.InPosFlapUpper;
      L     2;
      ==I;
      =     #FlapUpper.CmdMiddle1;
      L     #Ma.InPosFlapUpper;
      L     3;
      ==I;
      =     #FlapUpper.CmdHN;
//--- Sieve----
      AN    #LS1Sieve.StFault;
      AN    #LS2Sieve.StFault;
      A     #tmpEnable;
      =     #MotorSieve.InEnableFwd;
      A     #tmpNext;
      S     #MotorSieve.CmdNext;
      A     #tmpSeqStop;
      =     #MotorSieve.InSeqStop;
NETWORK
TITLE = temporare bits for Vendor
//--- Way Sieve Adjusted ---
      A(;
      A(;
      L     #Ma.InPosFlapLower;
      L     1;
      ==I;
      A     #FlapLower.StLN;
      );
      O(;
      L     #Ma.InPosFlapLower;
      L     2;
      ==I;
      A     #FlapLower.StMiddle1;
      );
      O(;
      L     #Ma.InPosFlapLower;
      L     3;
      ==I;
      A     #FlapLower.StHN;
      );
      ON    #Ma.Par.ParWithFlapLower;
      );
      A(;
      A(;
      L     #Ma.InPosFlapUpper;
      L     1;
      ==I;
      A     #FlapUpper.StLN;
      );
      O(;
      L     #Ma.InPosFlapUpper;
      L     2;
      ==I;
      A     #FlapUpper.StMiddle1;
      );
      O(;
      L     #Ma.InPosFlapUpper;
      L     3;
      ==I;
      A     #FlapUpper.StHN;
      );
      ON    #Ma.Par.ParWithFlapUpper;
      );
      =     #tmpWaySieveAdjusted;
//--- Enable Vendor----
      A     #tmpWaySieveAdjusted;
      A     #MotorSieve.StStartedFwd;
      ON    #Ma.Par.ParWithSieve;
      A     #tmpEnable;
      =     #tmpEnableVender;
//--Flap Vendor Adjusted
      A     #PosFlapAir.StMiddle1;
      ON    #Ma.Par.ParWithFlapAir;
      A(;
      A     #PosFlapFeed.StMiddle1;
      ON    #Ma.Par.ParWithFlapFeed;
      );
      =     #tmpFlapVendorAdjusted;
NETWORK
TITLE = Position AirFlap
      L     #Ma.Par.tmpPosFlapAir;
      L     #Ma.InPosFlapAirNom;
      T     #Ma.Par.tmpPosFlapAir;
      <>I;
      O     #Ma.CmdNewJob;
      JCN   FAJ2;
      R     #Ma.OutFlapAirLocal;
      A     #Ma.InAirRegulation;
      JC    FAJ2;
      L     #Ma.InPosFlapAirNom;
      DTR;
      T     #Ma.Par.OutPosFlapAirNom;
FAJ2: A     #Ma.InpAirMinus;
      O     #Ma.InpAirPlus;
      S     #Ma.OutFlapAirLocal;
//---Regulation of FlapAir-----
      A     #Ma.OutFlapAirLocal;
      ON    #Ma.InAirRegulation;
      ON    #Ma.Par.ParWithFlapAir;
      ON    #Ma.Par.ParWithFlowdetector;
      JC    FAJ5;
//---Integral Regulator------
      AN    #FlowDetector.OutL;
      O     #FlowDetector.OutH;
      A     "GCS7_Gr_OutTick200ms";
      JCN   FALM;
      L     2.000000e+00;	//[0.2s * 0.1]
      L     #Ma.Par.ParTI;	//Ma.Par.ParTI* 0.1s]
      DTR;
      /R;
      T     #tmpFactor;
      L     #Ma.InOverflow;
      L     #Ma.OutOverflow;
      -D;
      DTR;
      L     #tmpFactor;
      *R;
      L     #Ma.Par.OutPosFlapAirNom;
      +R;
      T     #Ma.Par.OutPosFlapAirNom;
//---Check Limit---
FALM: L     #Ma.Par.OutPosFlapAirNom;
      L     #Ma.InPosFlapAirNom;
      DTR;
      <=R;
      JC    FAL1;
      T     #Ma.Par.OutPosFlapAirNom;
FAL1: L     #Ma.Par.OutPosFlapAirNom;
      L     #Ma.InPosFlapAirMin;
      DTR;
      >=R;
      JC    FAJ5;
      T     #Ma.Par.OutPosFlapAirNom;
//--Target Position --------------
FAJ5: A     #Ma.OutFlapAirLocal;
      JC    FAHA;
      L     #Ma.Par.OutPosFlapAirNom;
      RND+;
      JU    FAJ9;
FAHA: L     #PosFlapAir.OutPosition;
      DTR;
      T     #Ma.Par.OutPosFlapAirNom;
      L     #PosFlapAir.OutPosition;
FAJ9: T     #PosFlapAir.InPositionMiddle;
      L     #PosFlapAir.OutPosition;
      T     #Ma.OutPosFlapAir;
NETWORK
TITLE = Interlocking Venders
//--- Monitoring
      SET;
      S     #FlowDetector.Par.ParLimitsPc;
      =     #FlowDetector.InMonHH;
      A     #Ma.InModeWarning;
      =     #FlowDetector.Par.ParWarningHH;
      L     #Ma.InPosFlapAirMin;
      L     #PosFlapAir.Par.ParPositionTolerance;
      +I;
      L     #Ma.OutPosFlapAir;
      >=I;
      AN    #Ma.OutFlapAirLocal;
      A     #Ma.InAirRegulation;
      =     #FlowDetector.InMonH;
      =     #FlowDetector.Par.ParWarningH;
//Tolerance band ---
      L     #Ma.InOverflow;
      L     #Ma.InTolOverflow;
      -I;
      L     10;
      *I;
      T     #FlowDetector.Par.ParLimitL;
      L     #Ma.InOverflow;
      L     #Ma.InTolOverflow;
      +I;
      L     10;
      *I;
      T     #FlowDetector.Par.ParLimitH;
//-- Limit------
      L     #Ma.InLimitOverflowFault;
      L     10;
      *I;
      T     #FlowDetector.Par.ParLimitHH;
//-- Actual Overflow---
      L     #FlowDetector.OutValuePc;
      L     10;
      /I;
      T     #Ma.OutOverflow;
//---Warning-----
      A     #FlowDetector.OutWarning;
      =     #Ma.OutWarning;
//--- Airlock----
      A     #Fan2.StStartedFwd;
      ON    #Ma.Par.ParWithFan2;
      A     #Fan1.StStartedFwd;
      A     #tmpEnableVender;
      =     #Airlock.InEnableFwd;
      A     #tmpNext;
      S     #Airlock.CmdNext;
      A     #tmpSeqStop;
      =     #Airlock.InSeqStop;
//--- FeedRoll----
      A     #Airlock.InEnableFwd;
      =     #FeedRoll.InEnableFwd;
      A     #PosFlapAir.StMiddle1;
      ON    #Ma.Par.ParWithFlapAir;
      A     #tmpNext;
      S     #FeedRoll.CmdNext;
      A     #tmpSeqStop;
      =     #FeedRoll.InSeqStop;
//--- Fan----
      SET;
      =     #Fan1.InEnableFwd;
      =     #Fan2.InEnableFwd;
      A     #tmpNext;
      S     #Fan1.CmdNext;
      A     #tmpNext;
      A     #tmpEnableVender;
      A     #Fan1.StStartedFwd;
      S     #Fan2.CmdNext;
      AN    #tmpEnable;
      O     #tmpSeqStop;
      =     #Fan1.InSeqStop;
      =     #Fan2.InSeqStop;
//-----FlapAir-------------
      A     #Ma.InpAirMinus;
      =     #PosFlapAir.InLN;
      A     #Ma.InpAirPlus;
      =     #PosFlapAir.CmdHN;
      AN    #Ma.InpAirMinus;
      AN    #Ma.InpAirPlus;
      AN    #tmpLocal;
      =     #PosFlapAir.CmdMiddle1;
      A     #tmpLocal;
      AN    #Ma.InpAirMinus;
      AN    #Ma.InpAirPlus;
      O     #MotorFlapAir.StFault;
      =     #PosFlapAir.InLocal;
//---MotorFlapAir--------------
      A     #PosFlapAir.OutpLN;
      AN    #Ma.OutFlapAirLocal;
      O     #Ma.InpAirMinus;
      =     #MotorFlapAir.InEnableRev;
      A     #PosFlapAir.OutpHN;
      AN    #Ma.OutFlapAirLocal;
      O     #Ma.InpAirPlus;
      =     #MotorFlapAir.InEnableFwd;
      A     #MotorFlapAir.InEnableRev;
      O     #MotorFlapAir.InEnableFwd;
      S     #MotorFlapAir.CmdNext;
      A     #MotorFlapAir.InpRunFwd;
      AN    #MotorFlapAir.OutpRunFwd;
      O;
      A     #MotorFlapAir.InpRunRev;
      AN    #MotorFlapAir.OutpRunRev;
      O;
      A     #tmpLocal;
      AN    #Ma.InpAirMinus;
      AN    #Ma.InpAirPlus;
      =     #MotorFlapAir.InLocal;
//----FlapFeed--------------
      A     #Ma.InpFeedMinus;
      =     #PosFlapFeed.InLN;
      A     #Ma.InpFeedPlus;
      =     #PosFlapFeed.CmdHN;
      AN    #Ma.InpFeedMinus;
      AN    #Ma.InpFeedPlus;
      AN    #tmpLocal;
      =     #PosFlapFeed.CmdMiddle1;
      A     #tmpLocal;
      AN    #Ma.InpFeedMinus;
      AN    #Ma.InpFeedPlus;
      O     #MotorFlapFeed.StFault;
      =     #PosFlapFeed.InLocal;
      L     #Ma.Par.tmpPosFlapFeed;
      L     #Ma.InPosFlapFeed;
      T     #Ma.Par.tmpPosFlapFeed;
      <>I;
      O     #Ma.CmdNewJob;
      R     #Ma.OutFlapFeedLocal;
      A     #Ma.InpFeedMinus;
      O     #Ma.InpFeedPlus;
      S     #Ma.OutFlapFeedLocal;
      A     #Ma.OutFlapFeedLocal;
      L     #PosFlapFeed.OutPosition;
      JC    FFJ1;
      L     #Ma.InPosFlapFeed;
FFJ1: T     #PosFlapFeed.InPositionMiddle;
      L     #PosFlapFeed.OutPosition;
      T     #Ma.OutPosFlapFeed;
//---MotorFlapFeed--------------
      A     #PosFlapFeed.OutpLN;
      AN    #Ma.OutFlapFeedLocal;
      O     #Ma.InpFeedMinus;
      =     #MotorFlapFeed.InEnableRev;
      A     #PosFlapFeed.OutpHN;
      AN    #Ma.OutFlapFeedLocal;
      O     #Ma.InpFeedPlus;
      =     #MotorFlapFeed.InEnableFwd;
      A     #MotorFlapFeed.InEnableFwd;
      O     #MotorFlapFeed.InEnableRev;
      S     #MotorFlapFeed.CmdNext;
      A     #MotorFlapFeed.InpRunFwd;
      AN    #MotorFlapFeed.OutpRunFwd;
      O;
      A     #MotorFlapFeed.InpRunRev;
      AN    #MotorFlapFeed.OutpRunRev;
      O;
      A     #tmpLocal;
      AN    #Ma.InpFeedMinus;
      AN    #Ma.InpFeedPlus;
      =     #MotorFlapFeed.InLocal;
NETWORK
TITLE = Call LS1Sieve
      AN    #Ma.Par.ParWithSieve;
      JC    EL2;
      CALL  #LS1Sieve;
NETWORK
TITLE = Call LS2Sieve
EL2:  AN    #Ma.Par.ParWithSieve;
      JC    EL3;
      CALL  #LS2Sieve;
NETWORK
TITLE = Call FlapLower
EL3:  AN    #Ma.Par.ParWithSieve;
      ON    #Ma.Par.ParWithFlapLower;
      JC    EL4;
      CALL  #FlapLower;
NETWORK
TITLE = Call FlapUpper
EL4:  AN    #Ma.Par.ParWithSieve;
      ON    #Ma.Par.ParWithFlapUpper;
      JC    EL5;
      CALL  #FlapUpper;
NETWORK
TITLE = Call Sieve
EL5:  AN    #Ma.Par.ParWithSieve;
      JC    EL6;
      CALL  #MotorSieve;
NETWORK
TITLE = Call FlapAir
EL6:  AN    #Ma.Par.ParWithVentus;
      ON    #Ma.Par.ParWithFlapAir;
      JC    EL7;
      SET;
      S     #PosFlapAir.Par.ParAngle;
      CALL  #PosFlapAir;
      CALL  #MotorFlapAir;
NETWORK
TITLE = Call FlapFeed
EL7:  AN    #Ma.Par.ParWithVentus;
      ON    #Ma.Par.ParWithFlapFeed;
      JC    EL8;
      SET;
      S     #PosFlapFeed.Par.ParAngle;
      CALL  #PosFlapFeed;
      CALL  #MotorFlapFeed;
NETWORK
TITLE = Call FlapFeedRoll
EL8:  AN    #Ma.Par.ParWithVentus;
      JC    EL9;
      CALL  #FeedRoll;
NETWORK
TITLE = Call Airlock
EL9:  AN    #Ma.Par.ParWithVentus;
      JC    EL10;
      CALL  #Airlock;
NETWORK
TITLE = Call Feedroll
EL10: AN    #Ma.Par.ParWithVentus;
      JC    EL11;
      CALL  #FeedRoll;
NETWORK
TITLE = Call Flowdetector
EL11: AN    #Ma.Par.ParWithVentus;
      ON    #Ma.Par.ParWithFlowdetector;
      JC    EL12;
      CALL  #FlowDetector;
NETWORK
TITLE = Call Fan1
EL12: AN    #Ma.Par.ParWithVentus;
      JC    EL13;
      CALL  #Fan1;
NETWORK
TITLE = Call Fan2
EL13: AN    #Ma.Par.ParWithVentus;
      ON    #Ma.Par.ParWithFan2;
      JC    EL14;
      CALL  #Fan2;
EL14: NOP   0;
NETWORK
TITLE = Temporare State bits
//---tmpStarted----
      A     #MotorSieve.StStartedFwd;
      ON    #Ma.Par.ParWithSieve;
      A(;
      A     #Airlock.StStartedFwd;
      ON    #Ma.Par.ParWithVentus;
      );
      A(;
      A     #FeedRoll.StStartedFwd;
      ON    #Ma.Par.ParWithVentus;
      );
      A     #tmpWaySieveAdjusted;
      =     #tmpStarted;
//---tmpStopped
      A     #MotorSieve.StStopped;
      ON    #Ma.Par.ParWithSieve;
      A(;
      A     #Airlock.StStopped;
      ON    #Ma.Par.ParWithVentus;
      );
      A(;
      A     #FeedRoll.StStopped;
      ON    #Ma.Par.ParWithVentus;
      );
      A(;
      A     #Fan1.StStopped;
      ON    #Ma.Par.ParWithVentus;
      );
      A(;
      A     #Fan2.StStopped;
      ON    #Ma.Par.ParWithFan2;
      );
      =     #tmpStopped;
NETWORK
TITLE = Jump to actual state
      A     #Ma.StStopped;
      JC    S0;	// ===> State
      A     #Ma.StStarted;
      JC    S2;	// ===> State
      A     #Ma.StStarting;
      JC    S1;	// ===> State
      A     #Ma.StStopping;
      JC    S3;	// ===> State
      A     #Ma.StClearing;
      JC    S5;	// ===> State
      A     #Ma.StFault;
      JC    S4;	// ===> State
NETWORK
TITLE = Stopped
xxS0: S     #Ma.StStopped;
S0:   A     #tmpFaultSum;
      R     #Ma.StStopped;
      JC    xxS4;	//--> StFault
      AN    #tmpStopped;
      R     #Ma.StStopped;
      JC    xxS1;	//--> StStarting
      JU    OUT;
NETWORK
TITLE = Starting
xxS1: S     #Ma.StStarting;
S1:   A     #tmpFaultSum;
      R     #Ma.StStarting;
      JC    xxS4;	//--> StFault
// Condition for StStopping
      AN    #tmpEnable;
      O     #tmpStopped;
      R     #Ma.StStarting;
      JC    xxS3;	//--> StStopping
// Condition for StStarted
      A     #tmpFlapVendorAdjusted;
      A     #tmpStarted;
      R     #Ma.StStarting;
      JC    xxS2;	//--> StStarted
      JU    OUT;
NETWORK
TITLE = Started
xxS2: S     #Ma.StStarted;
S2:   A     #tmpFaultSum;
      R     #Ma.StStarted;
      JC    xxS4;	//--> StFault
// Condition for StStopping
      AN    #tmpStarted;
      R     #Ma.StStarted;
      JC    xxS3;	//--> StStopping
// Condition for StClearing
      A     #Ma.InClearing;
      R     #Ma.StStarted;
      JC    xxS5;	//--> StClearing
      JU    OUT;
NETWORK
TITLE = StClearing
//any Transition 
xxS5: S     #Ma.StClearing;
      L     #Ma.Par.ParClearingTime;
      T     #Ma.Par.OutClearingTime;
//=== Logic
// Condition for StFault
S5:   A     #tmpFaultSum;
      R     #Ma.StClearing;
      JC    xxS4;	//--> StFault
// Condition for StStopping
      AN    #tmpStarted;
      R     #Ma.StClearing;
      JC    xxS3;	//--> StStopping
// Condition for StStarted
      AN    #Ma.InClearing;
      R     #Ma.StClearing;
      JC    xxS2;	//--> StStarted
      ON    "GCS7_Gr_OutTick500ms";	//Gr.OutTick500ms
      JC    OUT;
      L     #Ma.Par.OutClearingTime;
      +     -5;
      T     #Ma.Par.OutClearingTime;
      L     0;
      <=I;
      S     #Ma.OutCleared;
      JU    OUT;
NETWORK
TITLE = Stopping
xxS3: S     #Ma.StStopping;
S3:   A     #tmpFaultSum;
      R     #Ma.StStopping;
      JC    xxS4;	//--> StFault
// Condition for StStopped
      A     #tmpStopped;
      R     #Ma.StStopping;
      JC    xxS0;	//--> StStopped
// Condition for StStarting
      AN    #tmpSeqStop;
      O     #Ma.InManual;
      A     #tmpEnable;
      R     #Ma.StStopping;
      JC    xxS1;	//--> StStarting
      JU    OUT;
NETWORK
TITLE = Fault
xxS4: S     #Ma.StFault;
S4:   AN    #tmpFaultSum;
      R     #Ma.StFault;
      JC    xxS3;	//--> StStopping
      JU    OUT;
NETWORK
TITLE = Global End
OUT:  CLR;	//---Clear all commands
      =     #Ma.CmdOn;
      =     #Ma.CmdOff;
      =     #Ma.CmdNext;
      =     #Ma.CmdFaultReset;
      =     #Ma.CmdNewJob;
NETWORK
TITLE = State Code
// Same as Sieve
      L     32;	// StCode=Fault
      A     #Ma.StFault;
      JC    Code;
      L     1;	//StStopped
      A     #Ma.StStopped;
      JC    Code;
      L     2;	//StStarting
      A     #Ma.StStarting;
      JC    Code;
      L     13;	//StStarted.Warning
      A     #Ma.OutWarning;
      A     #Ma.StStarted;
      JC    Code;
      L     23;	//StStarted.Hand
      A     #Ma.OutFlapAirLocal;
      O     #Ma.OutFlapFeedLocal;
      A     #Ma.StStarted;
      JC    Code;
      L     3;	//StStarted
      A     #Ma.StStarted;
      JC    Code;
      L     7;	//StStopping
      A     #Ma.StStopping;
      JC    Code;
      L     8;	//StCode=Clearing
      A     #Ma.StClearing;
      JC    Code;
      L     32;	//StFault
Code: L     #Ma.StCode;	// Old state code
      TAK;
      T     #Ma.StCode;	// Save state code
      <>I;
      L     3;
      CC    "SYS_CBitCtrl";	//Set change bit
END_FUNCTION_BLOCK

FUNCTION_BLOCK "GCS7_M_FluidlifVessel"	// FB 82
TITLE = Pressure Vessel Conveying system
//  
//COPYRIGHT:    (C) 1999  BUEHLER AG, CH-9240 UZWIL, SWITZERLAND
//
//PRODUCT:      GCS7
//
//TITLE:        FB 82 Machine Control:Fluidlift with Vessel
//             
//GCPROVB:      Revision 11
//-------------------------------------------------------------------------
//
//IDENT:        AUTHOR:             DEPT:                       DATE:
//
//FB82.2.0      A. Egli             CT3                         15-Jul-2008
//              ParClearingPulseXxx
//FB82.1.1      A. Egli             CT3                          3-Mar-2005
//              Close Blowoff valve when stopped
//FB82.1.0      A. Egli             CT3                         15-Dec-2004
//              1st Release
//
//-------------------------------------------------------------------------
//
//PURPOSE:      MANUAL : see [LL.FLVxxMAN]
//
//RESTRICTIONS: S7
//-------------------------------------------------------------------------
//
AUTHOR : EA
FAMILY : GCS7LL
NAME : FLVessel
VERSION : 2.0
VAR
  Ma : UDT 20820;
  Blower : FB 12;
  Pressure : FB 16;
  BlowOff : FB 13;	//Element
  FillingFlap : FB 13;	//Element
  BlowlineFlap : FB 13;	//Element
  InletFlap : FB 13;	//Element
  OutletFlap : FB 13;	//Element
END_VAR
VAR_TEMP
  tmpEnable : BOOL ;
  tmpVKE : BOOL ;
  tmpEnableConveying : BOOL ;	//General condition for conveying Valve
  tmpLenDyn : INT ;
  tmpEnableClearing : BOOL ;
  tmpEnableFilling : BOOL ;
  tmpFillingReq : BOOL ;
  tmpFault : BOOL ;
  tmpLocal : BOOL ;
END_VAR
BEGIN
NETWORK
TITLE =
      L     30;
      T     #tmpLenDyn;
NETWORK
TITLE = PC Control
//=== Test Object number =====================
      L     "SYS_DirectCtrlDB".PC.ObjectNo;	//PCControl.ObjectNo
      L     #Ma.Par.ParObjectNo;	//Input ObjectNo
      <>I;
      JC    aEnd;
//=== Test OType      ========================
      L     2082;	//Input object type
      L     "SYS_DirectCtrlDB".PC.ObjectType;	//PCControl.ObjectType
      <>I;
      JC    aEnd;
//=== Test Handshake =========================
      A     "SYS_DirectCtrlDB".PC.Hsk.FExamine;	// Handshake.FExamine
      JC    aExa;
      A     "SYS_DirectCtrlDB".PC.Hsk.FDefineCmd;	// Handshake.FDefineCmd
      JC    aCmd;
      A     "SYS_DirectCtrlDB".PC.Hsk.FDefinePara;	// Handshake.FDefinePara
      JC    pPar;
aIni: L     2;	// FcInit
      UC    "SYS_DirectCtrl";
      JU    aEnd;
// Write parameter 
pPar: LAR1  P#DBX 58.0;
      L     P#6.0;
      +AR1;
      L     DBW [AR1,P#6.0];
      T     #Ma.Par.ParMinConveyingTime;
      L     DBW [AR1,P#8.0];
      T     #Ma.Par.ParClearingTime;
// Write new commands from PC to Interface of group 
aCmd: A     "SYS_DirectCtrlDB".PC.Cmd1[8];	//CmdOff   
      S     #Ma.CmdOff;
      A     "SYS_DirectCtrlDB".PC.Cmd1[9];	//CmdConveying
      S     #Ma.CmdConveying;
      A     "SYS_DirectCtrlDB".PC.Cmd1[10];	//CmdNext
      S     #Ma.CmdNext;
      A     "SYS_DirectCtrlDB".PC.Cmd1[11];	//CmdFaultReset
      S     #Ma.CmdFaultReset;
      A     "SYS_DirectCtrlDB".PC.Cmd1[14];	//CmdFilling
      S     #Ma.CmdFilling;
      A     "SYS_DirectCtrlDB".PC.Cmd1[13];	//CmdManualOn
      S     #Ma.InManual;
      A     "SYS_DirectCtrlDB".PC.Cmd2[13];	//CmdManualOff
      R     #Ma.InManual;
      JU    aIni;
aExa: TAR2;	// Address Dynamic datas
      T     "SYS_DirectCtrlDB".GC.InDynAddr;	// -->PCControl.GC.InDynAddr
      L     #tmpLenDyn;	// Length Dynamic datas
      T     "SYS_DirectCtrlDB".GC.InDynLen;	// -->PCControl.GC.InDynLen
      L     0;
      T     "SYS_DirectCtrlDB".GC.InParaAddr;	// -->PCControl.GC.InParaAddr
      T     "SYS_DirectCtrlDB".GC.InParaLen;	// -->PCControl.GC.InParaLen
      L     1;	// Code FcExamine
      UC    "SYS_DirectCtrl";
      L     11;	//Revision
      T     "SYS_DirectCtrlDB".GC.Revision;
aEnd: NOP   0;
NETWORK
TITLE = Interlocking
//===Global Group Orders===
//===Global Group Orders===
      A     "GCS7_Gr_OutManualOn";	///Gr.OutManualOn
      S     #Ma.InManual;
      A     "GCS7_Gr_OutManualOff";	//Gr.OutManualOff
      R     #Ma.InManual;
      A     #Ma.InManual;
      S     "GCS7_Gr_InManual";	//Gr.InManual
//Fault 
      O     #Blower.StFault;
      O     #Pressure.StFault;
      O     #BlowOff.StFault;
      O     #FillingFlap.StFault;
      O     #InletFlap.StFault;
      O     #BlowlineFlap.StFault;
      O     #OutletFlap.StFault;
      =     #tmpFault;
//Local
      A     #Ma.InLocal;
      AN    #Ma.InManual;
      =     #tmpLocal;
      A     #FillingFlap.StLN;
      ON    #Ma.Par.ParWithFillingFlap;
      A     #OutletFlap.StLN;
      A     #InletFlap.StLN;
      A     #BlowlineFlap.StLN;
      O     #tmpFault;
      A     #tmpLocal;
      S     #FillingFlap.InLocal;
      AN    #tmpLocal;
      R     #FillingFlap.InLocal;
      A     #FillingFlap.InLocal;
      =     #BlowlineFlap.InLocal;
      =     #InletFlap.InLocal;
      =     #OutletFlap.InLocal;
      A     #BlowOff.InLocal;	//[1.1]
      O     #BlowOff.StLN;	//[1.1]
      A     #FillingFlap.InLocal;	//[1.1]
      =     #BlowOff.InLocal;	//[1.1]
      A     #tmpLocal;
      =     #Blower.InLocal;
      =     #Pressure.InLocal;
//Enable 
      A(;
      AN    #Ma.InLocal;
      A     #Ma.InEnable;
      O;
      A     #Ma.OutManFilling;
      A     #Ma.InManual;
      O;
      A     #Ma.OutManConveying;
      A     #Ma.InManual;
      );
      AN    #Ma.CmdOff;
      =     #tmpEnable;
//Manual filling
      A     #Ma.CmdFilling;
      S     #Ma.OutManFilling;
      AN    #Ma.InManual;
      O     #Ma.CmdOff;
      O     #Ma.CmdConveying;
      R     #Ma.OutManFilling;
//Manual conveying
      A     #Ma.CmdConveying;
      S     #Ma.OutManConveying;
      AN    #Ma.InManual;
      O     #Ma.CmdOff;
      O     #Ma.CmdFilling;
      R     #Ma.OutManConveying;
//Warning
      A     #Pressure.OutNoMinP;
      =     #Ma.OutWarning;
NETWORK
TITLE = Call Blower
      CALL  #Blower;
NETWORK
TITLE = Call BlowOff
      CALL  #BlowOff;
NETWORK
TITLE = Call Pressure
      CALL  #Pressure;
NETWORK
TITLE = Call FillingFlap
      AN    #Ma.Par.ParWithFillingFlap;
      JC    E04;
      CALL  #FillingFlap;
NETWORK
TITLE = Call InletFlap
E04:  CALL  #InletFlap;
NETWORK
TITLE = Call BlowlineFlap
      CALL  #BlowlineFlap;
NETWORK
TITLE = Call OutletFlap
      CALL  #OutletFlap;
NETWORK
TITLE = Jump to actual state
      A     #Ma.StStopped;
      JC    S0;
      A     #Ma.StStarting;
      JC    S1;
      A     #Ma.StConveying;
      JC    S2;
      A     #Ma.StStopping;
      JC    S3;
      A     #Ma.StFault;
      JC    S4;
      A     #Ma.StClearing;
      JC    S5;
      A     #Ma.StWaiting;
      JC    S6;
      A     #Ma.StFilling;
      JC    S7;
      JU    xxS6;	// ===> Initialisation
NETWORK
TITLE = Stopped
//any Transition 
xxS0: S     #Ma.StStopped;
      JU    OUT;
//=== Logic
S0:   A     #tmpFault;
      R     #Ma.StStopped;
      JC    xxS4;	//-->Fault
      AN    #FillingFlap.StLN;
      A     #Ma.Par.ParWithFillingFlap;
      R     #Ma.StStopped;
      JC    xxS7;	//-->StFilling
      AN    #Blower.StStopped;
      AN    #Blower.StFault;
      R     #Ma.StStopped;
      JC    xxS1;	//-->Starting
      JU    OUT;
NETWORK
TITLE = StStarting
//any Transition 
xxS1: S     #Ma.StStarting;
//=== Logic
S1:   A     #tmpFault;
      R     #Ma.StStarting;
      JC    xxS4;	//-->Fault
      A     #Blower.StStopped;
      R     #Ma.StStarting;
      JC    xxS3;	//--> StStopping
      A     #Blower.StStartedFwd;
      R     #Ma.StStarting;
      JC    xxS6;
      JU    OUT;
NETWORK
TITLE = StConveying
//any Transition 
xxS2: S     #Ma.StConveying;
      R     #Ma.OutConveyingTimeDone;
      L     0;
      T     #Ma.Par.OutConveyingTime;
//=== Logic
// Condition for Stopped
S2:   A     #tmpFault;
      R     #Ma.StConveying;
      JC    xxS4;	//-->Fault
      AN    #Blower.StStartedFwd;
      R     #Ma.StConveying;
      JC    xxS3;	//--> StStopping
// Condition for Clearing
      AN    #OutletFlap.StHN;
      AN    #InletFlap.StHN;
      O     #Ma.OutConveyingTimeDone;
      R     #Ma.StConveying;
      JC    xxS5;	//--> StClearing
      A     #OutletFlap.StHN;
      A     #InletFlap.StHN;
      A     #BlowlineFlap.StHN;
      A     "GCS7_Gr_OutTick200ms";	//Gr.OutTick200ms
      JCN   S2H2;
      L     #Ma.Par.OutConveyingTime;
      +     2;
      T     #Ma.Par.OutConveyingTime;
      L     #Ma.Par.ParMinConveyingTime;
      L     #Ma.Par.OutConveyingTime;
      <=I;
      S     #Ma.OutConveyingTimeDone;
S2H2: JU    OUT;
NETWORK
TITLE = StStopping
//any Transition 
xxS3: S     #Ma.StStopping;
//=== Logic
S3:   A     #tmpFault;
      R     #Ma.StStopping;
      JC    xxS4;	//-->Fault
      A     #BlowOff.StLN;	//[1.1]
      ON    #Ma.InSeqStop;	//[1.1]
      A     #Blower.StStopped;
      R     #Ma.StStopping;
      JC    xxS0;	//--> StStopped
      JU    OUT;
NETWORK
TITLE = StFault
xxS4: S     #Ma.StFault;
S4:   A     #tmpFault;
      JC    OUT;
      A     #Blower.StStartedFwd;
      R     #Ma.StFault;
      JC    xxS6;	//--> StWaiting
      R     #Ma.StFault;
      JC    xxS3;	//--> StStopping
      JU    OUT;
NETWORK
TITLE = StClearing
//any Transition 
xxS5: S     #Ma.StClearing;
      R     #Ma.OutPulseOn;	//[2.0]
      L     0;
      T     #Ma.Par.OutClearingTime;
      L     #Ma.Par.ParClearingPulseOff;	//[2.0]
      T     #Ma.Par.OutPulseTime;	//[2.0]
//=== Logic
S5:   A     #tmpFault;
      R     #Ma.StClearing;
      R     #Ma.OutPulseOn;	//[2.0]
      JC    xxS4;	//-->Fault
// Condition for StCleared Case 1:
      L     #Ma.Par.ParClearingTime;
      L     #Ma.Par.OutClearingTime;
      <=I;
      A     #Ma.OutConveyingTimeDone;
      R     #Ma.OutLoaded;
// Condition for StStopped
      <=I;
//[2.0]      ON    #BlowlineFlap.StHN
      ON    #Blower.StStartedFwd;
      R     #Ma.StClearing;
      R     #Ma.OutPulseOn;	//[2.0]
      JC    xxS6;	//--> StWaiting
// Condition for StConveying
      A     #OutletFlap.StHN;
      A     #InletFlap.StHN;
      AN    #Ma.OutConveyingTimeDone;
      R     #Ma.StClearing;
      R     #Ma.OutPulseOn;	//[2.0]
      JC    xxS2;	//--> StConveing
//Pulse Time
      L     #Ma.Par.ParClearingPulseOff;	//[2.0]
      L     0;	//[2.0]
      ==I;	//[2.0]
      S     #Ma.OutPulseOn;	//[2.0]
      JC    S5CT;
      AN    "GCS7_Gr_OutTick200ms";	//[2.0]Gr.OutTick200ms
      JC    S5CT;
      L     #Ma.Par.OutPulseTime;	//[2.0]
      L     2;	//[2.0]
      -I;
      T     #Ma.Par.OutPulseTime;	//[2.0]
      JP    S5CT;	//[2.0]
      AN    #Ma.OutPulseOn;	//[2.0]
      =     #Ma.OutPulseOn;	//[2.0]
      L     #Ma.Par.ParClearingPulseOn;	//[2.0]
      JC    S5PT;	//[2.0]
      L     #Ma.Par.ParClearingPulseOff;	//[2.0]
S5PT: T     #Ma.Par.OutPulseTime;	//[2.0]
//Clearing Time                         //[2.0]
S5CT: AN    #Pressure.StMinP;	//[2.0]
      AN    #Ma.InNoWaitMinP;	//[2.0]
      L     0;	//[2.0]
      JC    S5C2;	//[2.0] -->Restart Clearing Time
      A     #Pressure.StMinP;
      O     #Ma.InNoWaitMinP;
      A     "GCS7_Gr_OutTick200ms";	//Gr.OutTick200ms
      AN    #tmpFault;
      JCN   OUT;
      L     #Ma.Par.OutClearingTime;
      +     2;
S5C2: T     #Ma.Par.OutClearingTime;
      JU    OUT;
NETWORK
TITLE = StWaiting
//any Transition 
xxS6: S     #Ma.StWaiting;
      JU    OUT;
//=== Logic
S6:   A     #tmpFault;	//-->StFault
      R     #Ma.StWaiting;
      JC    xxS4;
//Condition for StFilling
      AN    #FillingFlap.StLN;
      A     #Ma.Par.ParWithFillingFlap;
      R     #Ma.StWaiting;
      JC    xxS7;	//-->StFilling
//Condition for StConveying
      A     #OutletFlap.StHN;
      A     #InletFlap.StHN;
      A     #BlowlineFlap.StHN;
      A     #BlowOff.StLN;
      R     #Ma.StWaiting;
      JC    xxS2;	//-->StConveying
// Condition for StStopped
      AN    #Blower.StStartedFwd;
      R     #Ma.StWaiting;
      JC    xxS3;	//--> StStopping
      JU    OUT;
NETWORK
TITLE = StFilling
//any Transition 
xxS7: S     #Ma.StFilling;
      S     #Ma.OutLoaded;
      R     #Ma.OutConveyingTimeDone;
//=== Logic
S7:   A     #tmpFault;
      R     #Ma.StFilling;	//-->StFault
      JC    xxS4;
      A     #FillingFlap.StLN;
      R     #Ma.StFilling;
      JC    xxS6;	//--> StWaiting
      JU    OUT;
NETWORK
TITLE = State Code
// State           StCode
// ----------------------
// StFault            32
// StStopped.Empty     1
// StStopped.Loaded   11
// StStarting          2 
// StConveying         3
// StClearing.Ok       4
// StClearing.Warning 14
// StWaiting.Empty     6
// StWaiting.Loaded   16
// StStopping          7 
// StFilling           8
//
OUT:  L     1;	//Code=Stopped.Empty
      A     #Ma.StStopped;
      AN    #Ma.OutLoaded;
      JC    Code;
      L     11;	//Code=Stopped.Loaded
      A     #Ma.StStopped;
      JC    Code;
      L     2;	//Code=Staring
      A     #Ma.StStarting;
      JC    Code;
      L     3;	//Code=Conveying
      A     #Ma.StConveying;
      JC    Code;
      L     4;	//Code=Clearing.Ok
      A     #Ma.StClearing;
      AN    #Ma.OutWarning;
      JC    Code;
      L     14;	//Code=Clearing.Warning
      A     #Ma.StClearing;
      JC    Code;
      L     5;	//Code=Waiting.Empty
      A     #Ma.StWaiting;
      AN    #Ma.OutLoaded;
      JC    Code;
      L     15;	//Code=Waiting.Loaded
      A     #Ma.StWaiting;
      JC    Code;
      L     7;	//Code=Stopping
      A     #Ma.StStopping;
      JC    Code;
      L     8;	//Code=Filling
      A     #Ma.StFilling;
      JC    Code;
      L     32;	//StFault
Code: L     #Ma.StCode;	// Old state code
      TAK;
      T     #Ma.StCode;	// Save state code
      <>I;
      L     3;
      UC    "SYS_CBitCtrl";	//Set change bit
NETWORK
TITLE = General Commands
      A     #Ma.CmdFaultReset;
      S     #Blower.CmdFaultReset;
      S     #Pressure.CmdFaultReset;
      S     #BlowOff.CmdFaultReset;
      S     #FillingFlap.CmdFaultReset;
      S     #InletFlap.CmdFaultReset;
      S     #BlowlineFlap.CmdFaultReset;
      S     #OutletFlap.CmdFaultReset;
//----
      AN    #Ma.InManual;
      A     #Ma.InEnableFilling;
      O     #Ma.OutManFilling;
      =     #tmpFillingReq;
      A     #tmpFillingReq;
      A     #InletFlap.StLN;
      A     #OutletFlap.StLN;
      A     #BlowOff.StHN;
      =     #tmpEnableFilling;
//--- Manaul 
      A     #Ma.CmdConveying;
      A     #Ma.InManual;
      S     #Ma.OutLoaded;
      A     #Ma.OutManConveying;
      S     #Ma.CmdNext;
//---
      A     #Ma.OutLoaded;
      AN    #Ma.InManual;
      A(;
      AN    #Ma.OutConveyingTimeDone;
      ON    #Ma.InNoWaitMinP;
      ON    #Ma.OutLoaded;
      ON    #Ma.InEnableFilling;
      );
      O     #Ma.OutManConveying;
      A     #Blower.StStartedFwd;
      A(;
      A     #FillingFlap.StLN;
      ON    #Ma.Par.ParWithFillingFlap;
      );
      A     #tmpEnable;
      AN    #tmpLocal;
      =     #tmpEnableConveying;
NETWORK
TITLE = Commands Blower
      AN    #Pressure.StOverP;
      AN    #Pressure.StFault;
      AN    #BlowOff.StFault;
      A(;
      A     #InletFlap.StHN;
      AN    #BlowlineFlap.InManual;
      AN    #BlowlineFlap.StFault;
      O     #BlowOff.StHN;
      O     #BlowlineFlap.StHN;
      );
      A     #tmpEnable;
      AN    #Ma.StStopping;
      =     #Blower.InEnableFwd;
      A     #Blower.InEnableFwd;
      AN    #Blower.InSeqStop;
      AN    #BlowlineFlap.InManual;
      AN    #InletFlap.InManual;
      AN    #OutletFlap.InManual;
      AN    #tmpFault;
      A     #Ma.CmdNext;
      S     #Blower.CmdNext;
      AN    #Ma.OutLoaded;
      O     #tmpFault;
      O     #Ma.InSeqStop;
      =     #Blower.InSeqStop;
      A     #tmpFault;
      R     #Ma.OutAutostart;
      A     #Ma.CmdNext;
      O     #Ma.CmdConveying;
      S     #Ma.OutAutostart;
NETWORK
TITLE = Command FillingFlap
      A     #tmpEnableFilling;
      =     #FillingFlap.InEnableHN;
      NOT;
      =     #FillingFlap.InEnableLN;
      A     #Ma.CmdNext;
      O     #Ma.InManual;
      O     #FillingFlap.InEnableLN;
      S     #FillingFlap.CmdNext;
NETWORK
TITLE = Command BlowOffFlap
      A     #InletFlap.StHN;
      R     #BlowOff.InEnableHN;
      S     #BlowOff.InEnableLN;
      A     #Ma.StWaiting;
      A     #Ma.InClearing;
      ON    #tmpEnableConveying;
      ON    #Blower.StStartedFwd;
      ON    #FillingFlap.InEnableLN;
      S     #BlowOff.InEnableHN;
      R     #BlowOff.InEnableLN;
      A     #tmpLocal;	//[1.1]
      O     #Ma.InSeqStop;	//[1.1]
      A     #BlowlineFlap.StLN;	//[1.1]
      R     #BlowOff.InEnableHN;	//[1.1]
      S     #BlowOff.InEnableLN;	//[1.1]
      SET;
      S     #BlowOff.CmdNext;
NETWORK
TITLE = Command BlowLineFlap/ OutletFlap /InletFlap
//BlowlineFlap
      NOP   0;
//InletFlap   (Air)
      A     #tmpEnableConveying;
      S     #InletFlap.InEnableHN;
      R     #InletFlap.InEnableLN;
      AN    #tmpEnableConveying;
      A     #BlowOff.StHN;
      O     #Ma.InClearing;
      O     #Pressure.StCtoOverP;
      ON    #FillingFlap.InEnableLN;
      S     #InletFlap.InEnableLN;
      R     #InletFlap.InEnableHN;
      AN    #BlowlineFlap.InManual;
      AN    #OutletFlap.InManual;
      A     #Ma.CmdNext;
      O     #InletFlap.InEnableLN;
      S     #InletFlap.CmdNext;
//--OutletFlap ----
      A     #tmpEnableConveying;
      A     #BlowOff.StLN;
      S     #OutletFlap.InEnableHN;
      R     #OutletFlap.InEnableLN;
      AN    #tmpEnableConveying;
      A     #BlowOff.StHN;
      O     #Ma.InClearing;
      O     #Pressure.StCtoOverP;
      ON    #FillingFlap.InEnableLN;
      R     #OutletFlap.InEnableHN;
      S     #OutletFlap.InEnableLN;
      A     #OutletFlap.InEnableLN;
      AN    #OutletFlap.StLN;
      O     #Ma.OutAutostart;
      S     #OutletFlap.CmdNext;
//BlowlineFlap ----
      A     #tmpEnableConveying;
      A     #BlowOff.StLN;
      S     #BlowlineFlap.InEnableHN;
      R     #BlowlineFlap.InEnableLN;
      A     #Ma.InClearing;
      ON    #tmpEnableConveying;
      A     #BlowOff.StHN;
      O;
      AN    #Ma.OutPulseOn;	//[2.0]
      A     #Ma.StClearing;	//[2.0]
      A     #InletFlap.StHN;	//[2.0]
      ON    #FillingFlap.InEnableLN;
      R     #BlowlineFlap.InEnableHN;
      S     #BlowlineFlap.InEnableLN;
      A     #Ma.OutAutostart;
      O     #BlowlineFlap.InEnableLN;
      S     #BlowlineFlap.CmdNext;
NETWORK
TITLE = Interlocking Pressure
//--- Interlocking pressure 
      A     #Ma.StClearing;
      =     #Pressure.InMonMinP;
NETWORK
TITLE = Global End
//Next
//---Clear all commands
      CLR;
      =     #Ma.CmdOff;
      =     #Ma.CmdNext;
      =     #Ma.CmdFaultReset;
      =     #Ma.CmdConveying;
      =     #Ma.CmdFilling;
END_FUNCTION_BLOCK

FUNCTION_BLOCK "GCS7_E_Level"	// FB 84
TITLE = DigInpCont
//
//COPYRIGHT:    (C) 1996  BUHLER AG, CH-9240 UZWIL, SWITZERLAND
//
//PRODUCT:      GCS7
//
//TITLE:        Element Digital Input Continuous: SubType BinLevel
//
//-------------------------------------------------------------------------
//
//IDENT:        AUTHOR:             DEPT:                       DATE:
//FB84.1.0      A. Egli             CT3                         30-Oct-2002
//              SubType of FB14 Version 4.0
//
//-------------------------------------------------------------------------
//
//PURPOSE:      MANUAL : see [DICxxMAN]
//
//RESTRICTIONS: S7
//
//-------------------------------------------------------------------------
//
AUTHOR : EA
FAMILY : GCS90LL
NAME : DICLevel
VERSION : 1.0
VAR
  StCode : INT ;	//Element state code
  InMonCovered : BOOL ;	//After t4 must be in StCovered, otherwise it is a process fault
  InMonUncovered : BOOL ;	//After t5 must be in StUncovered, otherwise it is a process fault
  InPreAlarmCovered : BOOL ;	//LOG Pre-alarm if level is not covered
  InPreAlarmUncovered : BOOL ;	//LOG Pre-alarm if level is not uncovered
  InStopCoveredTime : BOOL ;	//Stop delay time t2
  InStopUncoveredTime : BOOL ;	//Stop delay time t3
  InpCovered : BOOL ;	//Digital input: 1=Covered , 0=Uncovered
  InpFaultDev : BOOL ;	//Digital input: fault device
  CmdRstCoveredTime : BOOL ;	//Restart delay time changing from Uncovered to Covered (t2)
  CmdRstUncoveredTime : BOOL ;	//Restart delay time changing from Covered to Uncovered (t3)
  CmdRunTimeoutTime : BOOL ;	//Run timeout time (only 1 working condition)
  CmdFaultReset : BOOL ;	//Command to reset fault
  InLocal : BOOL ;	//1= Local mode (automatic fault reset)
  spare0305 : BOOL ;
  InReport : BOOL ;	//Report of all state transitions
  OutTimeoutTime : BOOL ;	//Timeout time 1 working condition active
  InHWStop : BOOL ;	//HW stop is detected, no fault
  InDPFault : BOOL ;	//DP-Fault is detected, no fault
  OutPreAlarmCovered : BOOL ;	//Flag PreAlarmCovered is done
  OutPreAlarmUncovered : BOOL ;	//Flag PreAlarmUnCovered is done
  OutFlagPos : BOOL ;	//Positive flag InpCovered
  OutFlagNeg : BOOL ;	//Negative flag InpCovered
  OutpFaultReset : BOOL ;	//Reset alarm
  OutCovered : BOOL ;	//Copy of input signal
  StUncovered : BOOL ;	//Level is uncovered, delay time finished, monitoring is off
  StCtoCovered : BOOL ;	//Changing to Covered
  StCovered : BOOL ;	//Level is Covered, delay time finished
  StCtoUncovered : BOOL ;	//Changing to Uncovered
  StFault : BOOL ;	//Signal has not requested value, monitoring is active
  OutAlarmNrLog : INT ;	//Last textnumber send to log
  Par : STRUCT
   ParObjectNo : INT ;	//Is used for communication with PC, e.g. for message
   ParMsgType : INT ;	//Is used for message (translation of state)
   ParHornCode : INT ;	//Is used by horn module
   ParLogOff : BOOL ;	//Report is off
   spare0401 : BOOL ;
   Par2WorkingCond : BOOL ;	//Element has 2 defined working conditions
   ParFaultRetry : BOOL ;	//Retry after fault with monitoring- and delay-time
   ParBinLevel : BOOL ;	//Hold old state, if HWStop of DPFault
   ParDelayChange : INT ;	//Delay time, if the input changes, until the element changes its state
   ParDelayCovered : INT ;	//Time to change from StUncovered to StCovered
   ParDelayUncovered : INT ;	//Time to change from StCovered to StUncovered
   ParTimeoutCovered : INT ;	//If InMonCovered: after this time state has to be 'StCovered', otherwise StFault
   ParTimeoutUncovered : INT ;	//If InMonUncovered: after this time state has to be 'StUnCovered'
   OutMonTime : INT ;	//Actual time: monitoring
   OutTransitionTime : INT ;	//Actual time: changing state
   OutMonCovered : BOOL ;	//Monitoring time "Covered" is running
   OutMonUncovered : BOOL ;	//Monitoring time "Uncovered" is running
   OutFlagFaultDev : BOOL ;	//Flag InpFaultDev
   OutDelayTime : INT ;	//Actual time: DelayTime
  END_STRUCT ;
END_VAR
VAR_TEMP
  tmpLOGvalue : WORD ;	//LOG value
  tmpAddrPara : DWORD ;	//store the Instance Pointer
  tmpLenDyn : DINT ;
  tmpReport : BOOL ;	//Global LOG all
  tmpMonFault : BOOL ;	//Global monitor fault
  tmpMonOver : BOOL ;	//Monitoring time over
  tmp2WorkingCond : BOOL ;	//Monitoring time over
  tmpOutDelayDone : BOOL ;	//ParDelayTime Done
  tmpLocalFault : BOOL ;
  tmpLocal : BOOL ;
END_VAR
BEGIN
NETWORK
TITLE =
      UC    "GCS7_E_DigInput";
END_FUNCTION_BLOCK

